C05472=1208.877,279.801,-65.738,-176.741,6.965,148.342
C05473=1208.880,279.552,-65.710,-176.743,6.963,148.342
C05474=1208.885,279.304,-65.681,-176.745,6.959,148.342
C05475=1208.889,279.056,-65.652,-176.748,6.958,148.342
C05476=1208.894,278.808,-65.624,-176.751,6.955,148.342
C05477=1208.898,278.559,-65.596,-176.753,6.952,148.342
C05478=1208.903,278.311,-65.567,-176.755,6.950,148.342
C05479=1208.907,278.063,-65.539,-176.758,6.947,148.342
C05480=1208.912,277.814,-65.511,-176.760,6.945,148.342
C05481=1208.915,277.566,-65.483,-176.763,6.942,148.343
C05482=1208.920,277.318,-65.455,-176.766,6.940,148.343
C05483=1208.924,277.069,-65.426,-176.768,6.938,148.343
C05484=1208.929,276.821,-65.398,-176.770,6.935,148.343
C05485=1208.933,276.572,-65.370,-176.773,6.933,148.343
C05486=1208.937,276.324,-65.342,-176.776,6.930,148.343
C05487=1208.941,276.076,-65.314,-176.778,6.928,148.343
C05488=1208.946,275.828,-65.285,-176.780,6.926,148.344
C05489=1208.950,275.579,-65.257,-176.783,6.923,148.344
C05490=1208.955,275.330,-65.230,-176.785,6.921,148.344
C05491=1208.959,275.082,-65.201,-176.788,6.918,148.344
C05492=1208.963,274.834,-65.174,-176.791,6.916,148.344
C05493=1208.968,274.585,-65.145,-176.793,6.914,148.344
C05494=1208.972,274.337,-65.117,-176.796,6.911,148.344
C05495=1208.976,274.088,-65.089,-176.798,6.909,148.344
C05496=1208.981,273.840,-65.061,-176.801,6.906,148.345
C05497=1208.985,273.592,-65.033,-176.803,6.904,148.345
C05498=1208.990,273.343,-65.005,-176.805,6.902,148.345
C05499=1208.995,273.095,-64.977,-176.809,6.899,148.345
C05500=1208.998,272.846,-64.949,-176.811,6.897,148.345
C05501=1209.003,272.599,-64.921,-176.813,6.895,148.345
C05502=1209.007,272.350,-64.893,-176.816,6.892,148.346
C05503=1209.012,272.101,-64.865,-176.818,6.890,148.346
C05504=1209.016,271.853,-64.837,-176.821,6.887,148.346
C05505=1209.020,271.605,-64.809,-176.824,6.885,148.346
C05506=1209.025,271.357,-64.781,-176.826,6.883,148.346
C05507=1209.029,271.107,-64.754,-176.829,6.880,148.346
C05508=1209.033,270.859,-64.726,-176.831,6.878,148.346
C05509=1209.038,270.612,-64.698,-176.834,6.876,148.347
C05510=1209.042,270.362,-64.671,-176.836,6.873,148.347
C05511=1209.047,270.114,-64.642,-176.838,6.871,148.347
C05512=1209.051,269.866,-64.614,-176.841,6.869,148.347
C05513=1209.055,269.617,-64.587,-176.844,6.866,148.347
C05514=1209.060,269.369,-64.559,-176.846,6.864,148.347
C05515=1209.064,269.120,-64.532,-176.849,6.861,148.347
C05516=1209.069,268.872,-64.504,-176.851,6.859,148.347
C05517=1209.073,268.624,-64.476,-176.854,6.857,148.348
C05518=1209.077,268.375,-64.448,-176.856,6.854,148.348
C05519=1209.082,268.127,-64.421,-176.859,6.852,148.348
C05520=1209.086,267.878,-64.393,-176.861,6.850,148.348
C05521=1209.090,267.630,-64.365,-176.864,6.847,148.348
C05522=1209.095,267.381,-64.338,-176.867,6.845,148.349
C05523=1209.100,267.133,-64.310,-176.869,6.843,148.349
C05524=1209.104,266.885,-64.282,-176.872,6.840,148.349
C05525=1209.108,266.636,-64.255,-176.874,6.838,148.349
C05526=1209.113,266.388,-64.228,-176.877,6.836,148.349
C05527=1209.117,266.139,-64.200,-176.879,6.833,148.349
C05528=1209.121,265.890,-64.172,-176.882,6.831,148.350
C05529=1209.126,265.643,-64.145,-176.884,6.829,148.350
C05530=1209.130,265.394,-64.118,-176.887,6.826,148.350
C05531=1209.134,265.146,-64.089,-176.889,6.824,148.350
C05532=1209.139,264.897,-64.062,-176.891,6.822,148.350
C05533=1209.144,264.649,-64.034,-176.895,6.819,148.350
C05534=1209.148,264.400,-64.007,-176.897,6.817,148.350
C05535=1209.152,264.151,-63.980,-176.899,6.815,148.351
C05536=1209.157,263.903,-63.952,-176.902,6.813,148.351
C05537=1209.161,263.655,-63.925,-176.905,6.810,148.351
C05538=1209.165,263.382,-63.895,-176.907,6.808,148.351
C05539=1209.171,263.109,-63.864,-176.910,6.806,148.351
C05540=1209.175,262.837,-63.835,-176.913,6.803,148.352
C05541=1209.180,262.564,-63.804,-176.915,6.801,148.352
C05542=1209.185,262.316,-63.777,-176.919,6.798,148.352
C05543=1209.189,262.067,-63.750,-176.921,6.796,148.352
C05544=1209.194,261.818,-63.723,-176.923,6.794,148.352
C05545=1209.198,261.570,-63.695,-176.926,6.791,148.352
C05546=1209.203,261.322,-63.668,-176.929,6.789,148.353
C05547=1209.207,261.072,-63.640,-176.931,6.787,148.353
C05548=1209.211,260.824,-63.614,-176.933,6.785,148.353
C05549=1209.215,260.576,-63.586,-176.936,6.782,148.353
C05550=1209.220,260.328,-63.559,-176.939,6.780,148.353
C05551=1209.224,260.079,-63.532,-176.941,6.778,148.354
C05552=1209.229,259.831,-63.505,-176.944,6.775,148.354
C05553=1209.233,259.582,-63.478,-176.946,6.773,148.354
C05554=1209.238,259.334,-63.450,-176.949,6.771,148.354
C05555=1209.242,259.085,-63.423,-176.951,6.769,148.354
C05556=1209.247,258.837,-63.396,-176.954,6.766,148.355
C05557=1209.251,258.589,-63.369,-176.956,6.764,148.355
C05558=1209.255,258.340,-63.342,-176.959,6.762,148.355
C05559=1209.259,258.091,-63.315,-176.962,6.759,148.355
C05560=1209.264,257.842,-63.288,-176.964,6.757,148.355
C05561=1209.269,257.594,-63.261,-176.966,6.755,148.355
C05562=1209.273,257.346,-63.234,-176.969,6.753,148.356
C05563=1209.277,257.097,-63.207,-176.972,6.750,148.356
C05564=1209.282,256.849,-63.180,-176.974,6.748,148.356
C05565=1209.287,256.600,-63.153,-176.976,6.746,148.356
C05566=1209.291,256.351,-63.126,-176.979,6.744,148.356
C05567=1209.295,256.103,-63.098,-176.982,6.741,148.356
C05568=1209.299,255.854,-63.072,-176.984,6.740,148.357
C05569=1209.304,255.606,-63.045,-176.987,6.738,148.357
C05570=1209.309,255.357,-63.018,-176.989,6.735,148.357
C05571=1209.313,255.109,-62.991,-176.992,6.733,148.357
C05572=1209.317,254.861,-62.964,-176.994,6.731,148.358
C05573=1209.322,254.612,-62.937,-176.997,6.729,148.358
C05574=1209.327,254.364,-62.910,-177.000,6.726,148.358
C05575=1209.331,254.115,-62.883,-177.002,6.724,148.358
C05576=1209.335,253.867,-62.857,-177.004,6.722,148.358
C05577=1209.340,253.619,-62.830,-177.007,6.720,148.359
C05578=1209.344,253.369,-62.802,-177.010,6.718,148.359
C05579=1209.348,253.121,-62.776,-177.012,6.715,148.359
C05580=1209.352,252.873,-62.749,-177.015,6.713,148.359
C05581=1209.357,252.624,-62.722,-177.017,6.711,148.359
C05582=1209.361,252.375,-62.696,-177.020,6.709,148.360
C05583=1209.366,252.127,-62.669,-177.022,6.706,148.360
C05584=1209.371,251.878,-62.642,-177.025,6.704,148.360
C05585=1209.375,251.630,-62.615,-177.028,6.702,148.360
C05586=1209.379,251.381,-62.589,-177.030,6.700,148.360
C05587=1209.384,251.133,-62.562,-177.033,6.697,148.361
C05588=1209.388,250.884,-62.535,-177.035,6.695,148.361
C05589=1209.393,250.636,-62.508,-177.038,6.693,148.361
C05590=1209.397,250.387,-62.483,-177.040,6.691,148.361
C05591=1209.402,250.139,-62.456,-177.043,6.689,148.361
C05592=1209.406,249.890,-62.429,-177.046,6.687,148.362
C05593=1209.410,249.642,-62.402,-177.048,6.684,148.362
C05594=1209.415,249.393,-62.376,-177.051,6.683,148.362
C05595=1209.419,249.145,-62.349,-177.053,6.680,148.362
C05596=1209.424,248.896,-62.322,-177.056,6.678,148.363
C05597=1209.428,248.647,-62.296,-177.058,6.676,148.363
C05598=1209.433,248.399,-62.269,-177.061,6.674,148.363
C05599=1209.436,248.151,-62.243,-177.063,6.672,148.363
C05600=1209.441,247.902,-62.217,-177.065,6.670,148.363
C05601=1209.446,247.653,-62.189,-177.069,6.667,148.364
C05602=1209.450,247.404,-62.164,-177.071,6.665,148.364
C05603=1209.455,247.156,-62.137,-177.073,6.663,148.364
C05604=1209.460,246.908,-62.111,-177.076,6.661,148.364
C05605=1209.464,246.659,-62.084,-177.078,6.659,148.364
C05606=1209.468,246.411,-62.058,-177.081,6.656,148.365
C05607=1209.473,246.162,-62.031,-177.084,6.654,148.365
C05608=1209.477,245.914,-62.005,-177.086,6.652,148.365
C05609=1209.482,245.665,-61.979,-177.089,6.650,148.365
C05610=1209.486,245.416,-61.952,-177.091,6.648,148.366
C05611=1209.490,245.168,-61.926,-177.094,6.645,148.366
C05612=1209.495,244.919,-61.899,-177.097,6.644,148.366
C05613=1209.499,244.670,-61.874,-177.099,6.642,148.366
C05614=1209.504,244.422,-61.847,-177.101,6.640,148.367
C05615=1209.508,244.173,-61.821,-177.104,6.638,148.367
C05616=1209.513,243.926,-61.795,-177.107,6.635,148.367
C05617=1209.518,243.676,-61.768,-177.109,6.633,148.367
C05618=1209.522,243.428,-61.743,-177.112,6.631,148.368
C05619=1209.527,243.179,-61.715,-177.114,6.629,148.368
C05620=1209.531,242.930,-61.690,-177.117,6.627,148.368
C05621=1209.535,242.682,-61.663,-177.119,6.625,148.368
C05622=1209.540,242.433,-61.637,-177.122,6.622,148.368
C05623=1209.544,242.185,-61.612,-177.125,6.620,148.369
C05624=1209.548,241.937,-61.585,-177.127,6.618,148.369
C05625=1209.553,241.688,-61.559,-177.129,6.616,148.369
C05626=1209.558,241.439,-61.533,-177.132,6.614,148.369
C05627=1209.561,241.191,-61.507,-177.135,6.613,148.370
C05628=1209.566,240.941,-61.480,-177.137,6.609,148.370
C05629=1209.571,240.693,-61.455,-177.140,6.608,148.370
C05630=1209.575,240.445,-61.429,-177.143,6.606,148.370
C05631=1209.580,240.196,-61.402,-177.145,6.604,148.370
C05632=1209.584,239.947,-61.376,-177.147,6.602,148.371
C05633=1209.589,239.698,-61.350,-177.150,6.600,148.371
C05634=1209.593,239.450,-61.325,-177.153,6.597,148.371
C05635=1209.598,239.202,-61.298,-177.155,6.595,148.371
C05636=1209.602,238.953,-61.272,-177.158,6.593,148.372
C05637=1209.607,238.704,-61.247,-177.160,6.591,148.372
C05638=1209.611,238.455,-61.221,-177.163,6.589,148.372
C05639=1209.616,238.207,-61.195,-177.165,6.587,148.372
C05640=1209.620,237.959,-61.168,-177.168,6.585,148.373
C05641=1209.624,237.710,-61.143,-177.171,6.582,148.373
C05642=1209.629,237.438,-61.115,-177.173,6.581,148.373
C05643=1209.634,237.168,-61.086,-177.176,6.579,148.374
C05644=1209.640,236.895,-61.058,-177.179,6.576,148.374
C05645=1209.645,236.624,-61.030,-177.182,6.574,148.374
C05646=1209.649,236.375,-61.004,-177.184,6.572,148.374
C05647=1209.653,236.127,-60.978,-177.187,6.569,148.374
C05648=1209.657,235.878,-60.952,-177.190,6.568,148.375
C05649=1209.662,235.630,-60.926,-177.192,6.565,148.375
C05650=1209.666,235.381,-60.901,-177.195,6.563,148.375
C05651=1209.671,235.132,-60.874,-177.197,6.562,148.376
C05652=1209.675,234.884,-60.849,-177.200,6.560,148.376
C05653=1209.680,234.635,-60.823,-177.202,6.558,148.376
C05654=1209.685,234.387,-60.798,-177.205,6.556,148.376
C05655=1209.689,234.138,-60.772,-177.208,6.553,148.377
C05656=1209.694,233.890,-60.746,-177.210,6.551,148.377
C05657=1209.698,233.641,-60.721,-177.213,6.549,148.377
C05658=1209.702,233.392,-60.695,-177.215,6.547,148.377
C05659=1209.707,233.144,-60.669,-177.218,6.545,148.378
C05660=1209.712,232.895,-60.643,-177.220,6.543,148.378
C05661=1209.716,232.645,-60.618,-177.223,6.541,148.378
C05662=1209.721,232.397,-60.592,-177.225,6.539,148.378
C05663=1209.725,232.149,-60.567,-177.228,6.538,148.379
C05664=1209.730,231.900,-60.541,-177.231,6.535,148.379
C05665=1209.734,231.652,-60.516,-177.233,6.533,148.379
C05666=1209.739,231.403,-60.490,-177.236,6.531,148.379
C05667=1209.743,231.154,-60.464,-177.239,6.529,148.380
C05668=1209.748,230.906,-60.439,-177.241,6.527,148.380
C05669=1209.752,230.657,-60.414,-177.243,6.525,148.380
C05670=1209.756,230.408,-60.388,-177.246,6.523,148.380
C05671=1209.761,230.160,-60.363,-177.249,6.521,148.381
C05672=1209.766,229.911,-60.337,-177.251,6.519,148.381
C05673=1209.770,229.662,-60.311,-177.253,6.517,148.381
C05674=1209.775,229.413,-60.287,-177.257,6.515,148.382
C05675=1209.779,229.164,-60.261,-177.259,6.513,148.382
C05676=1209.784,228.916,-60.235,-177.262,6.511,148.382
C05677=1209.788,228.668,-60.210,-177.264,6.509,148.382
C05678=1209.793,228.418,-60.185,-177.267,6.507,148.383
C05679=1209.798,228.170,-60.159,-177.269,6.505,148.383
C05680=1209.801,227.922,-60.134,-177.272,6.503,148.383
C05681=1209.806,227.673,-60.109,-177.274,6.501,148.383
C05682=1209.810,227.424,-60.084,-177.277,6.499,148.384
C05683=1209.815,227.175,-60.058,-177.279,6.497,148.384
C05684=1209.819,226.927,-60.033,-177.282,6.496,148.384
C05685=1209.824,226.678,-60.008,-177.285,6.493,148.385
C05686=1209.829,226.430,-59.982,-177.287,6.491,148.385
C05687=1209.833,226.181,-59.956,-177.290,6.489,148.385
C05688=1209.838,225.932,-59.932,-177.293,6.487,148.385
C05689=1209.842,225.684,-59.907,-177.295,6.485,148.386
C05690=1209.847,225.435,-59.882,-177.298,6.483,148.386
C05691=1209.851,225.186,-59.856,-177.300,6.481,148.386
C05692=1209.856,224.938,-59.831,-177.303,6.479,148.386
C05693=1209.860,224.689,-59.806,-177.305,6.477,148.387
C05694=1209.865,224.440,-59.780,-177.308,6.476,148.387
C05695=1209.869,224.191,-59.756,-177.310,6.474,148.387
C05696=1209.873,223.942,-59.730,-177.313,6.472,148.388
C05697=1209.878,223.694,-59.705,-177.315,6.470,148.388
C05698=1209.883,223.445,-59.680,-177.318,6.468,148.388
C05699=1209.888,223.196,-59.655,-177.321,6.465,148.388
C05700=1209.891,222.948,-59.630,-177.324,6.463,148.389
C05701=1209.896,222.699,-59.605,-177.326,6.461,148.389
C05702=1209.900,222.450,-59.580,-177.329,6.459,148.389
C05703=1209.906,222.201,-59.555,-177.331,6.458,148.390
C05704=1209.909,221.953,-59.530,-177.334,6.456,148.390
C05705=1209.914,221.704,-59.505,-177.336,6.454,148.390
C05706=1209.919,221.456,-59.480,-177.339,6.452,148.391
C05707=1209.924,221.207,-59.455,-177.341,6.450,148.391
C05708=1209.928,220.958,-59.431,-177.344,6.448,148.391
C05709=1209.932,220.710,-59.405,-177.347,6.446,148.391
C05710=1209.937,220.461,-59.380,-177.349,6.444,148.392
C05711=1209.941,220.212,-59.356,-177.352,6.442,148.392
C05712=1209.946,219.964,-59.330,-177.354,6.441,148.392
C05713=1209.950,219.714,-59.305,-177.357,6.439,148.393
C05714=1209.955,219.466,-59.281,-177.359,6.437,148.393
C05715=1209.959,219.217,-59.255,-177.362,6.435,148.393
C05716=1209.964,218.968,-59.231,-177.364,6.433,148.393
C05717=1209.969,218.720,-59.207,-177.368,6.430,148.394
C05718=1209.973,218.471,-59.181,-177.370,6.428,148.394
C05719=1209.978,218.222,-59.156,-177.373,6.427,148.394
C05720=1209.982,217.973,-59.132,-177.376,6.425,148.395
C05721=1209.987,217.724,-59.107,-177.378,6.423,148.395
C05722=1209.991,217.477,-59.082,-177.380,6.421,148.395
C05723=1209.996,217.227,-59.057,-177.383,6.419,148.395
C05724=1210.001,216.979,-59.033,-177.386,6.417,148.396
C05725=1210.004,216.729,-59.008,-177.388,6.415,148.396
C05726=1210.010,216.481,-58.984,-177.391,6.413,148.396
C05727=1210.014,216.233,-58.959,-177.394,6.412,148.397
C05728=1210.018,215.983,-58.934,-177.396,6.409,148.397
C05729=1210.023,215.735,-58.909,-177.398,6.408,148.397
C05730=1210.028,215.486,-58.885,-177.401,6.406,148.398
C05731=1210.032,215.237,-58.860,-177.404,6.404,148.398
C05732=1210.037,214.988,-58.836,-177.406,6.402,148.398
C05733=1210.041,214.740,-58.810,-177.409,6.400,148.399
C05734=1210.045,214.491,-58.786,-177.412,6.398,148.399
C05735=1210.050,214.243,-58.761,-177.414,6.396,148.399
C05736=1210.055,213.994,-58.737,-177.417,6.395,148.400
C05737=1210.059,213.745,-58.712,-177.420,6.393,148.400
C05738=1210.064,213.496,-58.688,-177.422,6.391,148.400
C05739=1210.069,213.248,-58.663,-177.424,6.389,148.400
C05740=1210.073,212.998,-58.639,-177.427,6.387,148.401
C05741=1210.078,212.750,-58.614,-177.430,6.385,148.401
C05742=1210.082,212.501,-58.590,-177.432,6.383,148.401
C05743=1210.087,212.252,-58.565,-177.435,6.381,148.402
C05744=1210.091,212.003,-58.541,-177.438,6.380,148.402
C05745=1210.096,211.755,-58.517,-177.440,6.378,148.402
C05746=1210.101,211.485,-58.490,-177.443,6.375,148.403
C05747=1210.105,211.214,-58.463,-177.446,6.373,148.403
C05748=1210.111,210.943,-58.437,-177.449,6.371,148.403
C05749=1210.116,210.673,-58.411,-177.451,6.370,148.404
C05750=1210.120,210.425,-58.387,-177.454,6.368,148.404
C05751=1210.125,210.175,-58.362,-177.457,6.366,148.404
C05752=1210.129,209.927,-58.337,-177.459,6.364,148.405
C05753=1210.134,209.678,-58.313,-177.462,6.362,148.405
C05754=1210.139,209.430,-58.289,-177.464,6.360,148.405
C05755=1210.142,209.181,-58.264,-177.467,6.359,148.406
C05756=1210.147,208.932,-58.241,-177.470,6.357,148.406
C05757=1210.152,208.683,-58.216,-177.472,6.355,148.406
C05758=1210.157,208.434,-58.192,-177.475,6.353,148.407
C05759=1210.160,208.185,-58.168,-177.477,6.351,148.407
C05760=1210.166,207.937,-58.143,-177.480,6.349,148.407
C05761=1210.170,207.688,-58.119,-177.483,6.347,148.408
C05762=1210.175,207.439,-58.096,-177.485,6.345,148.408
C05763=1210.180,207.190,-58.071,-177.488,6.344,148.408
C05764=1210.184,206.941,-58.047,-177.490,6.342,148.409
C05765=1210.188,206.693,-58.022,-177.493,6.340,148.409
C05766=1210.193,206.444,-57.998,-177.496,6.338,148.409
C05767=1210.198,206.195,-57.974,-177.498,6.336,148.410
C05768=1210.202,205.947,-57.950,-177.501,6.334,148.410
C05769=1210.207,205.698,-57.926,-177.504,6.333,148.410
C05770=1210.211,205.448,-57.902,-177.506,6.331,148.411
C05771=1210.216,205.200,-57.878,-177.509,6.329,148.411
C05772=1210.220,204.951,-57.854,-177.512,6.327,148.411
C05773=1210.225,204.702,-57.830,-177.514,6.325,148.412
C05774=1210.230,204.454,-57.806,-177.517,6.323,148.412
C05775=1210.234,204.205,-57.781,-177.519,6.321,148.412
C05776=1210.239,203.956,-57.758,-177.522,6.319,148.412
C05777=1210.243,203.707,-57.734,-177.524,6.318,148.413
C05778=1210.247,203.459,-57.710,-177.527,6.316,148.413
C05779=1210.253,203.209,-57.686,-177.530,6.314,148.413
C05780=1210.257,202.961,-57.662,-177.532,6.313,148.414
C05781=1210.262,202.712,-57.638,-177.534,6.311,148.414
C05782=1210.266,202.464,-57.614,-177.537,6.309,148.414
C05783=1210.270,202.214,-57.591,-177.540,6.307,148.415
C05784=1210.275,201.965,-57.567,-177.542,6.306,148.415
C05785=1210.280,201.717,-57.542,-177.545,6.304,148.415
C05786=1210.285,201.468,-57.519,-177.548,6.302,148.416
C05787=1210.289,201.219,-57.494,-177.550,6.300,148.416
C05788=1210.294,200.970,-57.471,-177.553,6.298,148.417
C05789=1210.298,200.722,-57.447,-177.556,6.296,148.417
C05790=1210.303,200.473,-57.424,-177.558,6.295,148.417
C05791=1210.307,200.224,-57.400,-177.561,6.293,148.418
C05792=1210.312,199.975,-57.376,-177.563,6.291,148.418
C05793=1210.316,199.726,-57.352,-177.566,6.289,148.418
C05794=1210.321,199.477,-57.328,-177.569,6.287,148.419
C05795=1210.326,199.228,-57.304,-177.571,6.286,148.419
C05796=1210.330,198.979,-57.280,-177.573,6.284,148.419
C05797=1210.335,198.730,-57.257,-177.576,6.283,148.420
C05798=1210.339,198.482,-57.233,-177.579,6.281,148.420
C05799=1210.344,198.233,-57.210,-177.581,6.279,148.420
C05800=1210.349,197.984,-57.186,-177.584,6.277,148.421
C05801=1210.353,197.735,-57.162,-177.587,6.275,148.421
C05802=1210.358,197.486,-57.139,-177.589,6.273,148.421
C05803=1210.363,197.237,-57.115,-177.592,6.272,148.422
C05804=1210.367,196.989,-57.091,-177.595,6.270,148.422
C05805=1210.372,196.740,-57.068,-177.597,6.268,148.422
C05806=1210.376,196.491,-57.045,-177.600,6.266,148.423
C05807=1210.381,196.242,-57.021,-177.602,6.265,148.423
C05808=1210.385,195.993,-56.997,-177.605,6.263,148.423
C05809=1210.390,195.744,-56.974,-177.607,6.262,148.424
C05810=1210.394,195.496,-56.950,-177.610,6.260,148.424
C05811=1210.399,195.247,-56.926,-177.613,6.258,148.424
C05812=1210.404,194.998,-56.903,-177.615,6.256,148.425
C05813=1210.409,194.749,-56.880,-177.618,6.254,148.425
C05814=1210.413,194.500,-56.856,-177.621,6.252,148.426
C05815=1210.418,194.251,-56.832,-177.623,6.251,148.426
C05816=1210.422,194.002,-56.809,-177.625,6.250,148.426
C05817=1210.426,193.754,-56.786,-177.628,6.248,148.427
C05818=1210.431,193.505,-56.763,-177.631,6.246,148.427
C05819=1210.435,193.256,-56.739,-177.633,6.244,148.427
C05820=1210.440,193.007,-56.715,-177.636,6.242,148.428
C05821=1210.445,192.758,-56.692,-177.639,6.240,148.428
C05822=1210.450,192.509,-56.669,-177.641,6.239,148.428
C05823=1210.455,192.261,-56.646,-177.644,6.237,148.429
C05824=1210.460,192.012,-56.622,-177.646,6.236,148.429
C05825=1210.464,191.763,-56.599,-177.649,6.234,148.430
C05826=1210.468,191.514,-56.576,-177.652,6.232,148.430
C05827=1210.473,191.266,-56.552,-177.654,6.231,148.430
C05828=1210.477,191.017,-56.529,-177.657,6.229,148.431
C05829=1210.482,190.768,-56.505,-177.660,6.227,148.431
C05830=1210.487,190.519,-56.482,-177.662,6.225,148.431
C05831=1210.491,190.270,-56.459,-177.665,6.223,148.432
C05832=1210.495,190.021,-56.436,-177.667,6.222,148.432
C05833=1210.500,189.772,-56.413,-177.670,6.221,148.432
C05834=1210.505,189.523,-56.390,-177.672,6.219,148.433
C05835=1210.510,189.274,-56.366,-177.675,6.217,148.433
C05836=1210.514,189.026,-56.343,-177.678,6.215,148.434
C05837=1210.519,188.777,-56.320,-177.680,6.213,148.434
C05838=1210.523,188.528,-56.297,-177.683,6.211,148.434
C05839=1210.528,188.279,-56.273,-177.685,6.210,148.435
C05840=1210.533,188.030,-56.250,-177.688,6.209,148.435
C05841=1210.537,187.781,-56.227,-177.690,6.207,148.435
C05842=1210.542,187.532,-56.204,-177.694,6.205,148.436
C05843=1210.547,187.283,-56.182,-177.696,6.203,148.436
C05844=1210.551,187.034,-56.159,-177.699,6.202,148.437
C05845=1210.556,186.785,-56.135,-177.701,6.201,148.437
C05846=1210.560,186.536,-56.112,-177.704,6.199,148.437
C05847=1210.565,186.287,-56.089,-177.706,6.197,148.438
C05848=1210.570,186.039,-56.066,-177.709,6.195,148.438
C05849=1210.574,185.790,-56.043,-177.712,6.193,148.438
C05850=1210.580,185.520,-56.018,-177.714,6.192,148.439
C05851=1210.584,185.251,-55.994,-177.717,6.190,148.439
C05852=1210.590,184.981,-55.968,-177.720,6.188,148.440
C05853=1210.594,184.712,-55.944,-177.723,6.186,148.440
C05854=1210.599,184.462,-55.921,-177.725,6.185,148.440
C05855=1210.604,184.213,-55.897,-177.728,6.183,148.441
C05856=1210.608,183.964,-55.875,-177.731,6.181,148.441
C05857=1210.613,183.716,-55.852,-177.733,6.180,148.441
C05858=1210.618,183.467,-55.829,-177.736,6.178,148.442
C05859=1210.622,183.218,-55.806,-177.739,6.177,148.442
C05860=1210.627,182.968,-55.784,-177.741,6.175,148.443
C05861=1210.631,182.720,-55.761,-177.744,6.173,148.443
C05862=1210.636,182.471,-55.738,-177.746,6.172,148.443
C05863=1210.641,182.222,-55.714,-177.749,6.170,148.444
C05864=1210.645,181.973,-55.692,-177.751,6.168,148.444
C05865=1210.650,181.724,-55.669,-177.754,6.167,148.445
C05866=1210.654,181.476,-55.647,-177.757,6.165,148.445
C05867=1210.659,181.226,-55.624,-177.759,6.164,148.445
C05868=1210.663,180.978,-55.601,-177.762,6.162,148.446
C05869=1210.668,180.728,-55.578,-177.764,6.160,148.446
C05870=1210.673,180.480,-55.556,-177.767,6.159,148.447
C05871=1210.678,180.231,-55.533,-177.770,6.157,148.447
C05872=1210.682,179.981,-55.511,-177.772,6.156,148.447
C05873=1210.687,179.733,-55.488,-177.775,6.154,148.448
C05874=1210.691,179.484,-55.465,-177.777,6.152,148.448
C05875=1210.696,179.235,-55.442,-177.780,6.150,148.448
C05876=1210.701,178.987,-55.420,-177.783,6.149,148.449
C05877=1210.706,178.737,-55.397,-177.785,6.148,148.449
C05878=1210.710,178.488,-55.375,-177.788,6.146,148.450
C05879=1210.715,178.239,-55.352,-177.790,6.144,148.450
C05880=1210.719,177.991,-55.329,-177.793,6.142,148.450
C05881=1210.724,177.741,-55.307,-177.795,6.141,148.451
C05882=1210.728,177.492,-55.284,-177.798,6.140,148.451
C05883=1210.734,177.243,-55.262,-177.801,6.138,148.451
C05884=1210.738,176.995,-55.239,-177.804,6.136,148.452
C05885=1210.742,176.745,-55.217,-177.806,6.135,148.452
C05886=1210.747,176.497,-55.194,-177.808,6.134,148.453
C05887=1210.752,176.248,-55.172,-177.811,6.132,148.453
C05888=1210.756,175.999,-55.149,-177.814,6.130,148.454
C05889=1210.761,175.750,-55.127,-177.816,6.128,148.454
C05890=1210.765,175.501,-55.104,-177.818,6.127,148.454
C05891=1210.771,175.252,-55.082,-177.822,6.126,148.455
C05892=1210.775,175.003,-55.060,-177.824,6.124,148.455
C05893=1210.780,174.754,-55.036,-177.827,6.122,148.456
C05894=1210.785,174.505,-55.015,-177.829,6.121,148.456
C05895=1210.789,174.257,-54.992,-177.832,6.119,148.456
C05896=1210.794,174.007,-54.969,-177.834,6.117,148.457
C05897=1210.798,173.758,-54.948,-177.838,6.116,148.457
C05898=1210.802,173.510,-54.925,-177.840,6.115,148.458
C05899=1210.808,173.261,-54.903,-177.842,6.113,148.458
C05900=1210.812,173.011,-54.881,-177.845,6.111,148.458
C05901=1210.817,172.763,-54.858,-177.848,6.109,148.459
C05902=1210.822,172.514,-54.836,-177.850,6.109,148.459
C05903=1210.826,172.264,-54.814,-177.853,6.107,148.460
C05904=1210.831,172.016,-54.792,-177.855,6.105,148.460
C05905=1210.836,171.767,-54.768,-177.858,6.103,148.460
C05906=1210.841,171.518,-54.747,-177.860,6.102,148.461
C05907=1210.845,171.269,-54.725,-177.863,6.101,148.461
C05908=1210.850,171.020,-54.703,-177.866,6.099,148.462
C05909=1210.854,170.771,-54.680,-177.869,6.097,148.462
C05910=1210.859,170.522,-54.658,-177.871,6.096,148.463
C05911=1210.863,170.273,-54.636,-177.873,6.095,148.463
C05912=1210.868,170.024,-54.614,-177.876,6.093,148.463
C05913=1210.873,169.775,-54.592,-177.879,6.091,148.464
C05914=1210.878,169.525,-54.570,-177.881,6.090,148.464
C05915=1210.882,169.277,-54.547,-177.884,6.088,148.465
C05916=1210.886,169.028,-54.525,-177.887,6.087,148.465
C05917=1210.891,168.779,-54.503,-177.889,6.086,148.465
C05918=1210.896,168.530,-54.481,-177.891,6.084,148.466
C05919=1210.901,168.281,-54.459,-177.894,6.082,148.466
C05920=1210.905,168.032,-54.437,-177.897,6.081,148.467
C05921=1210.910,167.783,-54.415,-177.899,6.080,148.467
C05922=1210.915,167.534,-54.393,-177.902,6.078,148.467
C05923=1210.920,167.285,-54.370,-177.905,6.076,148.468
C05924=1210.924,167.036,-54.348,-177.907,6.075,148.468
C05925=1210.929,166.787,-54.327,-177.910,6.074,148.469
C05926=1210.933,166.538,-54.305,-177.913,6.072,148.469
C05927=1210.938,166.289,-54.283,-177.915,6.070,148.469
C05928=1210.942,166.040,-54.261,-177.917,6.069,148.470
C05929=1210.947,165.791,-54.239,-177.920,6.067,148.470
C05930=1210.952,165.542,-54.217,-177.923,6.066,148.471
C05931=1210.956,165.293,-54.195,-177.925,6.065,148.471
C05932=1210.962,165.044,-54.173,-177.928,6.063,148.472
C05933=1210.966,164.795,-54.151,-177.931,6.061,148.472
C05934=1210.971,164.547,-54.129,-177.933,6.060,148.472
C05935=1210.975,164.297,-54.107,-177.936,6.059,148.473
C05936=1210.980,164.049,-54.086,-177.939,6.057,148.473
C05937=1210.985,163.799,-54.064,-177.941,6.056,148.474
C05938=1210.990,163.550,-54.043,-177.943,6.054,148.474
C05939=1210.994,163.301,-54.021,-177.946,6.053,148.475
C05940=1210.999,163.052,-53.999,-177.949,6.051,148.475
C05941=1211.004,162.803,-53.977,-177.951,6.050,148.475
C05942=1211.008,162.554,-53.955,-177.954,6.048,148.476
C05943=1211.013,162.305,-53.934,-177.957,6.046,148.476
C05944=1211.017,162.056,-53.912,-177.959,6.045,148.477
C05945=1211.022,161.807,-53.890,-177.962,6.044,148.477
C05946=1211.027,161.558,-53.869,-177.965,6.042,148.477
C05947=1211.032,161.309,-53.847,-177.967,6.041,148.478
C05948=1211.036,161.060,-53.825,-177.970,6.039,148.478
C05949=1211.041,160.811,-53.803,-177.972,6.038,148.479
C05950=1211.046,160.562,-53.781,-177.975,6.037,148.479
C05951=1211.050,160.313,-53.760,-177.977,6.035,148.480
C05952=1211.055,160.064,-53.738,-177.980,6.033,148.480
C05953=1211.060,159.815,-53.717,-177.982,6.032,148.481
C05954=1211.065,159.546,-53.693,-177.985,6.031,148.481
C05955=1211.070,159.277,-53.670,-177.988,6.029,148.482
C05956=1211.075,159.008,-53.647,-177.991,6.027,148.482
C05957=1211.080,158.739,-53.624,-177.994,6.026,148.483
C05958=1211.085,158.490,-53.602,-177.996,6.025,148.483
C05959=1211.089,158.241,-53.580,-177.999,6.023,148.483
C05960=1211.094,157.991,-53.559,-178.002,6.021,148.484
C05961=1211.099,157.743,-53.537,-178.004,6.021,148.484
C05962=1211.103,157.493,-53.515,-178.007,6.019,148.485
C05963=1211.109,157.244,-53.494,-178.009,6.017,148.485
C05964=1211.113,156.996,-53.473,-178.012,6.016,148.485
C05965=1211.117,156.747,-53.451,-178.015,6.015,148.486
C05966=1211.122,156.497,-53.430,-178.017,6.013,148.486
C05967=1211.127,156.249,-53.409,-178.020,6.012,148.487
C05968=1211.132,156.000,-53.387,-178.023,6.010,148.487
C05969=1211.137,155.750,-53.366,-178.025,6.009,148.488
C05970=1211.141,155.501,-53.344,-178.027,6.008,148.488
C05971=1211.146,155.252,-53.323,-178.030,6.006,148.488
C05972=1211.150,155.003,-53.301,-178.033,6.005,148.489
C05973=1211.155,154.754,-53.280,-178.035,6.003,148.489
C05974=1211.160,154.505,-53.259,-178.038,6.002,148.490
C05975=1211.165,154.257,-53.237,-178.040,6.001,148.490
C05976=1211.169,154.007,-53.216,-178.043,5.999,148.491
C05977=1211.174,153.758,-53.195,-178.046,5.997,148.491
C05978=1211.179,153.509,-53.174,-178.048,5.996,148.492
C05979=1211.184,153.260,-53.152,-178.051,5.995,148.492
C05980=1211.188,153.011,-53.131,-178.053,5.994,148.493
C05981=1211.192,152.762,-53.110,-178.056,5.992,148.493
C05982=1211.198,152.513,-53.089,-178.059,5.990,148.493
C05983=1211.202,152.264,-53.067,-178.061,5.990,148.494
C05984=1211.207,152.015,-53.047,-178.064,5.988,148.494
C05985=1211.211,151.765,-53.025,-178.066,5.987,148.495
C05986=1211.216,151.517,-53.004,-178.069,5.985,148.495
C05987=1211.222,151.267,-52.983,-178.072,5.984,148.496
C05988=1211.226,151.019,-52.962,-178.074,5.983,148.496
C05989=1211.231,150.770,-52.941,-178.077,5.981,148.497
C05990=1211.235,150.520,-52.919,-178.079,5.980,148.497
C05991=1211.240,150.271,-52.898,-178.082,5.978,148.497
C05992=1211.245,150.022,-52.877,-178.085,5.977,148.498
C05993=1211.250,149.774,-52.855,-178.087,5.976,148.498
C05994=1211.254,149.525,-52.835,-178.090,5.974,148.499
C05995=1211.259,149.275,-52.814,-178.092,5.973,148.499
C05996=1211.263,149.026,-52.792,-178.095,5.972,148.500
C05997=1211.268,148.777,-52.772,-178.098,5.970,148.500
C05998=1211.273,148.528,-52.751,-178.100,5.969,148.501
C05999=1211.278,148.279,-52.729,-178.103,5.968,148.501
C06000=1211.282,148.030,-52.709,-178.105,5.967,148.502
C06001=1211.287,147.780,-52.687,-178.108,5.965,148.502
C06002=1211.292,147.531,-52.666,-178.111,5.963,148.503
C06003=1211.296,147.283,-52.645,-178.113,5.962,148.503
C06004=1211.301,147.033,-52.624,-178.116,5.961,148.503
C06005=1211.306,146.784,-52.604,-178.118,5.960,148.504
C06006=1211.311,146.535,-52.583,-178.121,5.958,148.504
C06007=1211.316,146.287,-52.561,-178.123,5.957,148.505
C06008=1211.320,146.038,-52.541,-178.126,5.956,148.505
C06009=1211.325,145.788,-52.520,-178.129,5.954,148.506
C06010=1211.329,145.539,-52.499,-178.131,5.953,148.506
C06011=1211.335,145.289,-52.478,-178.134,5.951,148.507
C06012=1211.339,145.041,-52.457,-178.136,5.951,148.507
C06013=1211.344,144.792,-52.436,-178.139,5.949,148.508
C06014=1211.348,144.543,-52.416,-178.142,5.948,148.508
C06015=1211.353,144.294,-52.395,-178.144,5.946,148.509
C06016=1211.358,144.045,-52.375,-178.147,5.945,148.509
C06017=1211.363,143.795,-52.354,-178.150,5.944,148.510
C06018=1211.368,143.547,-52.333,-178.152,5.942,148.510
C06019=1211.372,143.297,-52.312,-178.154,5.941,148.510
C06020=1211.376,143.048,-52.291,-178.158,5.940,148.511
C06021=1211.381,142.799,-52.270,-178.160,5.939,148.511
C06022=1211.386,142.550,-52.249,-178.162,5.937,148.512
C06023=1211.391,142.301,-52.228,-178.165,5.936,148.512
C06024=1211.395,142.052,-52.208,-178.168,5.934,148.513
C06025=1211.401,141.803,-52.187,-178.170,5.933,148.513
C06026=1211.405,141.554,-52.167,-178.173,5.932,148.514
C06027=1211.410,141.304,-52.146,-178.176,5.930,148.514
C06028=1211.415,141.055,-52.125,-178.178,5.929,148.515
C06029=1211.419,140.806,-52.105,-178.181,5.928,148.515
C06030=1211.424,140.557,-52.084,-178.183,5.927,148.516
C06031=1211.429,140.308,-52.064,-178.186,5.925,148.516
C06032=1211.434,140.059,-52.043,-178.188,5.924,148.517
C06033=1211.438,139.810,-52.022,-178.191,5.923,148.517
C06034=1211.443,139.561,-52.002,-178.194,5.922,148.518
C06035=1211.448,139.312,-51.981,-178.196,5.920,148.518
C06036=1211.452,139.063,-51.961,-178.198,5.919,148.518
C06037=1211.458,138.814,-51.940,-178.202,5.918,148.519
C06038=1211.462,138.565,-51.919,-178.204,5.916,148.519
C06039=1211.467,138.315,-51.900,-178.207,5.915,148.520
C06040=1211.472,138.066,-51.879,-178.209,5.914,148.520
C06041=1211.476,137.817,-51.858,-178.212,5.913,148.521
C06042=1211.481,137.568,-51.838,-178.215,5.911,148.521
C06043=1211.486,137.319,-51.817,-178.217,5.910,148.522
C06044=1211.490,137.070,-51.797,-178.220,5.908,148.522
C06045=1211.495,136.821,-51.776,-178.222,5.908,148.523
C06046=1211.500,136.571,-51.756,-178.225,5.906,148.523
C06047=1211.505,136.322,-51.736,-178.227,5.905,148.524
C06048=1211.509,136.073,-51.715,-178.230,5.904,148.524
C06049=1211.514,135.824,-51.694,-178.232,5.903,148.525
C06050=1211.519,135.575,-51.674,-178.235,5.901,148.525
C06051=1211.524,135.325,-51.654,-178.238,5.900,148.526
C06052=1211.528,135.076,-51.634,-178.241,5.899,148.526
C06053=1211.534,134.828,-51.613,-178.243,5.898,148.527
C06054=1211.538,134.579,-51.593,-178.245,5.896,148.527
C06055=1211.543,134.330,-51.573,-178.248,5.895,148.528
C06056=1211.548,134.080,-51.552,-178.251,5.894,148.528
C06057=1211.553,133.831,-51.532,-178.253,5.893,148.529
C06058=1211.557,133.562,-51.511,-178.256,5.891,148.529
C06059=1211.563,133.294,-51.488,-178.259,5.890,148.530
C06060=1211.568,133.024,-51.466,-178.261,5.889,148.530
C06061=1211.572,132.756,-51.445,-178.264,5.887,148.531
C06062=1211.577,132.507,-51.424,-178.267,5.886,148.531
C06063=1211.583,132.258,-51.404,-178.270,5.885,148.532
C06064=1211.587,132.009,-51.384,-178.272,5.883,148.532
C06065=1211.592,131.760,-51.364,-178.275,5.883,148.533
C06066=1211.597,131.511,-51.344,-178.277,5.882,148.533
C06067=1211.601,131.262,-51.324,-178.280,5.880,148.533
C06068=1211.607,131.012,-51.303,-178.282,5.879,148.534
C06069=1211.611,130.763,-51.283,-178.285,5.877,148.534
C06070=1211.615,130.514,-51.263,-178.288,5.877,148.535
C06071=1211.621,130.265,-51.243,-178.290,5.875,148.536
C06072=1211.625,130.016,-51.223,-178.293,5.874,148.536
C06073=1211.630,129.767,-51.203,-178.296,5.873,148.537
C06074=1211.634,129.518,-51.183,-178.298,5.872,148.537
C06075=1211.639,129.268,-51.163,-178.301,5.870,148.538
C06076=1211.644,129.019,-51.142,-178.303,5.869,148.538
C06077=1211.650,128.770,-51.123,-178.306,5.868,148.539
C06078=1211.654,128.521,-51.103,-178.308,5.867,148.539
C06079=1211.658,128.272,-51.082,-178.312,5.865,148.540
C06080=1211.663,128.022,-51.063,-178.314,5.865,148.540
C06081=1211.668,127.774,-51.042,-178.316,5.863,148.540
C06082=1211.673,127.525,-51.023,-178.319,5.862,148.541
C06083=1211.678,127.275,-51.003,-178.321,5.861,148.541
C06084=1211.682,127.026,-50.983,-178.324,5.860,148.542
C06085=1211.687,126.777,-50.963,-178.326,5.859,148.542
C06086=1211.691,126.528,-50.943,-178.330,5.857,148.543
C06087=1211.697,126.279,-50.924,-178.332,5.856,148.543
C06088=1211.701,126.030,-50.903,-178.335,5.855,148.544
C06089=1211.706,125.780,-50.884,-178.337,5.854,148.545
C06090=1211.710,125.531,-50.863,-178.340,5.852,148.545
C06091=1211.715,125.282,-50.843,-178.342,5.852,148.546
C06092=1211.720,125.033,-50.824,-178.345,5.850,148.546
C06093=1211.725,124.784,-50.804,-178.348,5.849,148.547
C06094=1211.730,124.534,-50.784,-178.350,5.848,148.547
C06095=1211.734,124.285,-50.765,-178.353,5.847,148.548
C06096=1211.739,124.037,-50.745,-178.355,5.846,148.548
C06097=1211.744,123.787,-50.725,-178.358,5.844,148.549
C06098=1211.749,123.537,-50.705,-178.360,5.843,148.549
C06099=1211.753,123.288,-50.685,-178.363,5.842,148.550
C06100=1211.759,123.040,-50.666,-178.366,5.841,148.550
C06101=1211.763,122.790,-50.646,-178.368,5.840,148.550
C06102=1211.768,122.541,-50.625,-178.371,5.839,148.551
C06103=1211.773,122.292,-50.606,-178.373,5.838,148.551
C06104=1211.778,122.043,-50.587,-178.376,5.836,148.552
C06105=1211.783,121.793,-50.567,-178.378,5.835,148.553
C06106=1211.787,121.544,-50.547,-178.381,5.834,148.553
C06107=1211.792,121.295,-50.527,-178.384,5.833,148.554
C06108=1211.797,121.046,-50.508,-178.386,5.832,148.554
C06109=1211.802,120.796,-50.488,-178.389,5.831,148.555
C06110=1211.806,120.548,-50.469,-178.391,5.830,148.555
C06111=1211.811,120.299,-50.449,-178.394,5.828,148.556
C06112=1211.816,120.049,-50.429,-178.397,5.828,148.556
C06113=1211.821,119.800,-50.410,-178.399,5.827,148.557
C06114=1211.826,119.551,-50.390,-178.402,5.825,148.557
C06115=1211.831,119.301,-50.371,-178.404,5.824,148.558
C06116=1211.836,119.053,-50.351,-178.407,5.823,148.558
C06117=1211.840,118.804,-50.332,-178.409,5.822,148.559
C06118=1211.844,118.554,-50.312,-178.413,5.820,148.559
C06119=1211.850,118.305,-50.293,-178.415,5.819,148.560
C06120=1211.854,118.056,-50.273,-178.417,5.819,148.560
C06121=1211.859,117.806,-50.253,-178.420,5.817,148.561
C06122=1211.865,117.557,-50.234,-178.423,5.816,148.561
C06123=1211.869,117.308,-50.215,-178.425,5.815,148.562
C06124=1211.874,117.059,-50.196,-178.428,5.814,148.562
C06125=1211.878,116.810,-50.175,-178.430,5.813,148.563
C06126=1211.883,116.560,-50.156,-178.433,5.812,148.564
C06127=1211.888,116.312,-50.136,-178.435,5.811,148.564
C06128=1211.892,116.062,-50.117,-178.438,5.810,148.565
C06129=1211.897,115.813,-50.098,-178.441,5.808,148.565
C06130=1211.902,115.564,-50.078,-178.443,5.808,148.566
C06131=1211.907,115.314,-50.059,-178.446,5.806,148.566
C06132=1211.912,115.066,-50.040,-178.449,5.805,148.567
C06133=1211.917,114.816,-50.020,-178.451,5.804,148.567
C06134=1211.922,114.567,-50.001,-178.454,5.803,148.568
C06135=1211.927,114.318,-49.981,-178.456,5.802,148.568
C06136=1211.931,114.068,-49.962,-178.459,5.801,148.569
C06137=1211.936,113.820,-49.943,-178.461,5.800,148.569
C06138=1211.941,113.570,-49.923,-178.464,5.799,148.570
C06139=1211.946,113.321,-49.905,-178.467,5.797,148.570
C06140=1211.950,113.071,-49.886,-178.469,5.797,148.571
C06141=1211.956,112.822,-49.866,-178.471,5.796,148.571
C06142=1211.960,112.573,-49.847,-178.475,5.794,148.572
C06143=1211.964,112.324,-49.828,-178.477,5.793,148.572
C06144=1211.970,112.075,-49.808,-178.480,5.792,148.573
C06145=1211.974,111.825,-49.789,-178.482,5.791,148.573
C06146=1211.979,111.577,-49.770,-178.485,5.790,148.574
C06147=1211.984,111.327,-49.750,-178.487,5.789,148.574
C06148=1211.989,111.078,-49.732,-178.490,5.788,148.575
C06149=1211.994,110.828,-49.713,-178.492,5.787,148.575
C06150=1211.999,110.579,-49.693,-178.495,5.786,148.576
C06151=1212.003,110.330,-49.674,-178.497,5.785,148.576
C06152=1212.008,110.081,-49.655,-178.500,5.784,148.577
C06153=1212.013,109.832,-49.635,-178.503,5.782,148.577
C06154=1212.018,109.583,-49.617,-178.505,5.782,148.578
C06155=1212.023,109.333,-49.598,-178.508,5.781,148.579
C06156=1212.027,109.084,-49.579,-178.511,5.779,148.579
C06157=1212.032,108.835,-49.559,-178.513,5.779,148.580
C06158=1212.037,108.586,-49.541,-178.516,5.777,148.580
C06159=1212.042,108.336,-49.522,-178.518,5.776,148.581
C06160=1212.047,108.087,-49.503,-178.521,5.775,148.581
C06161=1212.051,107.838,-49.483,-178.524,5.774,148.582
C06162=1212.057,107.569,-49.463,-178.526,5.773,148.583
C06163=1212.062,107.301,-49.442,-178.529,5.772,148.583
C06164=1212.067,107.033,-49.423,-178.532,5.771,148.584
C06165=1212.072,106.765,-49.402,-178.535,5.770,148.584
C06166=1212.077,106.515,-49.383,-178.537,5.769,148.585
C06167=1212.082,106.266,-49.365,-178.540,5.768,148.585
C06168=1212.087,106.016,-49.345,-178.542,5.766,148.586
C06169=1212.091,105.768,-49.326,-178.545,5.766,148.586
C06170=1212.096,105.518,-49.307,-178.548,5.765,148.587
C06171=1212.101,105.269,-49.289,-178.550,5.763,148.587
C06172=1212.106,105.019,-49.269,-178.553,5.763,148.588
C06173=1212.111,104.770,-49.251,-178.555,5.762,148.588
C06174=1212.116,104.521,-49.232,-178.558,5.760,148.589
C06175=1212.120,104.272,-49.213,-178.560,5.759,148.589
C06176=1212.126,104.023,-49.194,-178.563,5.759,148.590
C06177=1212.130,103.773,-49.175,-178.566,5.757,148.591
C06178=1212.135,103.524,-49.157,-178.568,5.757,148.591
C06179=1212.140,103.275,-49.138,-178.571,5.756,148.592
C06180=1212.144,103.025,-49.119,-178.573,5.755,148.592
C06181=1212.150,102.777,-49.100,-178.576,5.754,148.593
C06182=1212.154,102.527,-49.082,-178.578,5.753,148.593
C06183=1212.159,102.278,-49.062,-178.581,5.752,148.594
C06184=1212.164,102.029,-49.044,-178.584,5.750,148.594
C06185=1212.168,101.779,-49.025,-178.586,5.750,148.595
C06186=1212.174,101.530,-49.007,-178.589,5.749,148.596
C06187=1212.178,101.281,-48.988,-178.592,5.747,148.596
C06188=1212.183,101.031,-48.970,-178.594,5.747,148.597
C06189=1212.188,100.783,-48.951,-178.596,5.746,148.597
C06190=1212.192,100.533,-48.932,-178.599,5.744,148.598
C06191=1212.198,100.284,-48.913,-178.602,5.744,148.598
C06192=1212.203,100.035,-48.895,-178.604,5.743,148.599
C06193=1212.207,99.785,-48.877,-178.607,5.742,148.599
C06194=1212.212,99.536,-48.857,-178.610,5.740,148.600
C06195=1212.217,99.287,-48.839,-178.612,5.740,148.601
C06196=1212.221,99.038,-48.820,-178.614,5.739,148.601
C06197=1212.227,98.788,-48.802,-178.617,5.738,148.602
C06198=1212.232,98.539,-48.784,-178.620,5.737,148.602
C06199=1212.236,98.290,-48.765,-178.622,5.736,148.603
C06200=1212.241,98.040,-48.746,-178.625,5.735,148.603
C06201=1212.246,97.792,-48.727,-178.628,5.734,148.604
C06202=1212.251,97.542,-48.709,-178.630,5.733,148.604
C06203=1212.255,97.293,-48.691,-178.633,5.732,148.605
C06204=1212.261,97.044,-48.672,-178.635,5.731,148.605
C06205=1212.266,96.794,-48.654,-178.638,5.730,148.606
C06206=1212.270,96.545,-48.635,-178.640,5.729,148.606
C06207=1212.275,96.295,-48.617,-178.643,5.729,148.607
C06208=1212.280,96.047,-48.598,-178.646,5.727,148.608
C06209=1212.285,95.797,-48.580,-178.648,5.726,148.608
C06210=1212.289,95.548,-48.562,-178.651,5.726,148.609
C06211=1212.295,95.299,-48.543,-178.653,5.725,148.609
C06212=1212.300,95.049,-48.525,-178.656,5.723,148.610
C06213=1212.304,94.800,-48.506,-178.659,5.723,148.611
C06214=1212.309,94.550,-48.488,-178.661,5.722,148.611
C06215=1212.313,94.302,-48.470,-178.664,5.720,148.612
C06216=1212.319,94.052,-48.451,-178.667,5.720,148.612
C06217=1212.323,93.802,-48.433,-178.669,5.719,148.613
C06218=1212.328,93.553,-48.415,-178.671,5.718,148.613
C06219=1212.333,93.304,-48.397,-178.674,5.717,148.614
C06220=1212.338,93.056,-48.378,-178.677,5.716,148.614
C06221=1212.343,92.806,-48.360,-178.679,5.715,148.615
C06222=1212.348,92.556,-48.341,-178.681,5.714,148.615
C06223=1212.353,92.307,-48.323,-178.685,5.713,148.616
C06224=1212.358,92.058,-48.305,-178.687,5.712,148.616
C06225=1212.362,91.809,-48.287,-178.689,5.711,148.617
C06226=1212.367,91.559,-48.269,-178.692,5.711,148.618
C06227=1212.371,91.310,-48.250,-178.695,5.709,148.618
C06228=1212.377,91.061,-48.231,-178.697,5.709,148.619
C06229=1212.382,90.812,-48.213,-178.700,5.708,148.620
C06230=1212.387,90.562,-48.196,-178.702,5.707,148.620
C06231=1212.391,90.313,-48.177,-178.705,5.706,148.621
C06232=1212.396,90.063,-48.159,-178.708,5.705,148.621
C06233=1212.401,89.814,-48.141,-178.710,5.704,148.622
C06234=1212.406,89.565,-48.123,-178.713,5.704,148.622
C06235=1212.411,89.316,-48.105,-178.715,5.702,148.623
C06236=1212.416,89.067,-48.087,-178.718,5.701,148.623
C06237=1212.420,88.817,-48.069,-178.721,5.701,148.624
C06238=1212.425,88.568,-48.051,-178.723,5.700,148.624
C06239=1212.430,88.318,-48.033,-178.725,5.699,148.625
C06240=1212.436,88.069,-48.014,-178.729,5.698,148.626
C06241=1212.440,87.820,-47.996,-178.731,5.697,148.626
C06242=1212.445,87.571,-47.978,-178.733,5.696,148.627
C06243=1212.450,87.321,-47.960,-178.736,5.696,148.627
C06244=1212.455,87.072,-47.942,-178.739,5.694,148.628
C06245=1212.459,86.822,-47.924,-178.741,5.693,148.629
C06246=1212.464,86.573,-47.906,-178.743,5.692,148.629
C06247=1212.469,86.324,-47.888,-178.746,5.692,148.630
C06248=1212.474,86.075,-47.870,-178.749,5.691,148.630
C06249=1212.479,85.826,-47.852,-178.751,5.689,148.631
C06250=1212.484,85.576,-47.834,-178.754,5.689,148.631
C06251=1212.489,85.327,-47.816,-178.757,5.688,148.632
C06252=1212.494,85.077,-47.799,-178.759,5.687,148.632
C06253=1212.498,84.828,-47.781,-178.762,5.686,148.633
C06254=1212.503,84.578,-47.763,-178.765,5.685,148.634
C06255=1212.508,84.329,-47.745,-178.767,5.684,148.634
C06256=1212.512,84.080,-47.727,-178.769,5.684,148.635
C06257=1212.517,83.831,-47.709,-178.772,5.683,148.635
C06258=1212.522,83.582,-47.691,-178.775,5.681,148.636
C06259=1212.528,83.332,-47.674,-178.777,5.681,148.637
C06260=1212.532,83.083,-47.656,-178.780,5.680,148.637
C06261=1212.537,82.834,-47.638,-178.782,5.679,148.638
C06262=1212.542,82.585,-47.620,-178.785,5.679,148.638
C06263=1212.547,82.336,-47.602,-178.788,5.677,148.639
C06264=1212.552,82.086,-47.585,-178.790,5.676,148.639
C06265=1212.557,81.837,-47.567,-178.793,5.676,148.640
C06266=1212.562,81.568,-47.547,-178.795,5.675,148.641
C06267=1212.568,81.299,-47.529,-178.798,5.674,148.641
C06268=1212.573,81.031,-47.509,-178.801,5.673,148.642
C06269=1212.578,80.763,-47.490,-178.804,5.673,148.643
C06270=1212.583,80.513,-47.473,-178.806,5.671,148.643
C06271=1212.587,80.264,-47.455,-178.809,5.670,148.644
C06272=1212.592,80.015,-47.437,-178.812,5.670,148.644
C06273=1212.597,79.766,-47.419,-178.814,5.669,148.645
C06274=1212.602,79.516,-47.402,-178.816,5.668,148.645
C06275=1212.607,79.267,-47.384,-178.819,5.668,148.646
C06276=1212.612,79.018,-47.366,-178.822,5.666,148.646
C06277=1212.617,78.768,-47.349,-178.824,5.665,148.647
C06278=1212.622,78.519,-47.331,-178.827,5.665,148.648
C06279=1212.626,78.270,-47.314,-178.829,5.664,148.648
C06280=1212.632,78.020,-47.296,-178.832,5.663,148.649
C06281=1212.637,77.771,-47.278,-178.835,5.662,148.650
C06282=1212.641,77.522,-47.262,-178.837,5.661,148.650
C06283=1212.646,77.272,-47.244,-178.840,5.661,148.651
C06284=1212.651,77.023,-47.226,-178.842,5.660,148.651
C06285=1212.656,76.773,-47.208,-178.844,5.659,148.652
C06286=1212.661,76.524,-47.190,-178.847,5.658,148.652
C06287=1212.666,76.275,-47.174,-178.850,5.657,148.653
C06288=1212.670,76.026,-47.156,-178.853,5.656,148.654
C06289=1212.676,75.776,-47.138,-178.855,5.656,148.654
C06290=1212.680,75.527,-47.121,-178.858,5.655,148.655
C06291=1212.685,75.278,-47.103,-178.860,5.654,148.655
C06292=1212.690,75.028,-47.086,-178.862,5.653,148.656
C06293=1212.695,74.779,-47.068,-178.865,5.653,148.657
C06294=1212.700,74.530,-47.052,-178.868,5.652,148.657
C06295=1212.705,74.281,-47.034,-178.870,5.651,148.658
C06296=1212.710,74.031,-47.016,-178.873,5.650,148.658
C06297=1212.714,73.782,-46.999,-178.876,5.649,148.659
C06298=1212.719,73.532,-46.982,-178.878,5.649,148.660
C06299=1212.725,73.283,-46.964,-178.880,5.648,148.660
C06300=1212.730,73.033,-46.946,-178.884,5.647,148.661
C06301=1212.734,72.784,-46.930,-178.886,5.646,148.661
C06302=1212.739,72.535,-46.912,-178.888,5.645,148.662
C06303=1212.744,72.285,-46.895,-178.891,5.645,148.662
C06304=1212.748,72.036,-46.877,-178.894,5.644,148.663
C06305=1212.754,71.787,-46.860,-178.896,5.643,148.664
C06306=1212.759,71.537,-46.844,-178.898,5.642,148.664
C06307=1212.764,71.288,-46.826,-178.902,5.641,148.665
C06308=1212.769,71.038,-46.808,-178.904,5.640,148.665
C06309=1212.773,70.790,-46.791,-178.906,5.640,148.666
C06310=1212.778,70.540,-46.774,-178.909,5.639,148.667
C06311=1212.783,70.290,-46.756,-178.912,5.638,148.667
C06312=1212.788,70.041,-46.739,-178.914,5.638,148.668
C06313=1212.793,69.792,-46.722,-178.916,5.637,148.668
C06314=1212.798,69.543,-46.705,-178.919,5.636,148.669
C06315=1212.803,69.293,-46.687,-178.922,5.635,148.670
C06316=1212.808,69.044,-46.670,-178.924,5.634,148.670
C06317=1212.813,68.794,-46.654,-178.927,5.634,148.671
C06318=1212.817,68.545,-46.636,-178.930,5.633,148.671
C06319=1212.822,68.295,-46.619,-178.932,5.632,148.672
C06320=1212.828,68.046,-46.602,-178.934,5.631,148.672
C06321=1212.832,67.797,-46.585,-178.937,5.631,148.673
C06322=1212.837,67.548,-46.567,-178.940,5.630,148.674
C06323=1212.842,67.298,-46.551,-178.943,5.629,148.674
C06324=1212.847,67.048,-46.533,-178.945,5.628,148.675
C06325=1212.852,66.800,-46.517,-178.948,5.627,148.676
C06326=1212.857,66.550,-46.499,-178.950,5.627,148.676
C06327=1212.861,66.301,-46.482,-178.952,5.626,148.677
C06328=1212.867,66.051,-46.465,-178.955,5.625,148.677
C06329=1212.871,65.802,-46.449,-178.958,5.625,148.678
C06330=1212.877,65.553,-46.431,-178.960,5.624,148.679
C06331=1212.881,65.304,-46.414,-178.962,5.623,148.679
C06332=1212.886,65.054,-46.397,-178.966,5.622,148.680
C06333=1212.891,64.804,-46.380,-178.968,5.621,148.680
C06334=1212.896,64.555,-46.363,-178.971,5.621,148.681
C06335=1212.901,64.306,-46.347,-178.973,5.620,148.681
C06336=1212.906,64.056,-46.329,-178.976,5.619,148.682
C06337=1212.910,63.807,-46.312,-178.978,5.619,148.683
C06338=1212.916,63.557,-46.295,-178.981,5.618,148.683
C06339=1212.921,63.309,-46.279,-178.983,5.617,148.684
C06340=1212.925,63.059,-46.262,-178.986,5.617,148.685
C06341=1212.930,62.809,-46.245,-178.988,5.616,148.685
C06342=1212.935,62.560,-46.228,-178.991,5.616,148.686
C06343=1212.941,62.311,-46.211,-178.994,5.614,148.686
C06344=1212.945,62.061,-46.194,-178.996,5.613,148.687
C06345=1212.950,61.812,-46.177,-178.999,5.613,148.688
C06346=1212.955,61.562,-46.160,-179.002,5.612,148.688
C06347=1212.960,61.313,-46.144,-179.004,5.611,148.689
C06348=1212.965,61.063,-46.127,-179.006,5.611,148.689
C06349=1212.969,60.815,-46.109,-179.009,5.610,148.690
C06350=1212.974,60.566,-46.093,-179.012,5.610,148.691
C06351=1212.980,60.316,-46.076,-179.014,5.609,148.691
C06352=1212.984,60.067,-46.059,-179.016,5.608,148.692
C06353=1212.989,59.817,-46.042,-179.019,5.608,148.693
C06354=1212.995,59.567,-46.026,-179.022,5.607,148.693
C06355=1212.999,59.318,-46.010,-179.024,5.605,148.694
C06356=1213.004,59.068,-45.992,-179.027,5.605,148.694
C06357=1213.009,58.819,-45.976,-179.030,5.604,148.695
C06358=1213.014,58.570,-45.959,-179.032,5.604,148.696
C06359=1213.019,58.320,-45.942,-179.034,5.603,148.696
C06360=1213.024,58.071,-45.926,-179.037,5.602,148.697
C06361=1213.029,57.822,-45.909,-179.040,5.602,148.697
C06362=1213.033,57.572,-45.893,-179.042,5.601,148.698
C06363=1213.039,57.323,-45.876,-179.045,5.600,148.699
C06364=1213.044,57.074,-45.859,-179.047,5.600,148.699
C06365=1213.048,56.824,-45.842,-179.050,5.599,148.700
C06366=1213.054,56.575,-45.825,-179.052,5.598,148.700
C06367=1213.059,56.325,-45.809,-179.055,5.598,148.701
C06368=1213.063,56.075,-45.793,-179.057,5.597,148.702
C06369=1213.068,55.827,-45.777,-179.060,5.596,148.702
C06370=1213.074,55.558,-45.758,-179.063,5.595,148.703
C06371=1213.079,55.290,-45.740,-179.066,5.595,148.704
C06372=1213.084,55.022,-45.723,-179.068,5.594,148.704
C06373=1213.090,54.753,-45.704,-179.071,5.593,148.705
C06374=1213.095,54.504,-45.688,-179.074,5.593,148.706
C06375=1213.100,54.254,-45.672,-179.076,5.592,148.706
C06376=1213.104,54.004,-45.655,-179.078,5.591,148.707
C06377=1213.109,53.755,-45.639,-179.081,5.591,148.707
C06378=1213.114,53.506,-45.622,-179.084,5.589,148.708
C06379=1213.119,53.257,-45.606,-179.087,5.589,148.709
C06380=1213.124,53.007,-45.590,-179.089,5.588,148.709
C06381=1213.129,52.757,-45.573,-179.092,5.587,148.710
C06382=1213.134,52.509,-45.557,-179.094,5.587,148.710
C06383=1213.139,52.258,-45.540,-179.097,5.586,148.711
C06384=1213.144,52.009,-45.524,-179.100,5.586,148.712
C06385=1213.149,51.760,-45.507,-179.102,5.585,148.712
C06386=1213.153,51.510,-45.490,-179.104,5.584,148.713
C06387=1213.159,51.261,-45.475,-179.107,5.584,148.714
C06388=1213.163,51.011,-45.458,-179.110,5.583,148.714
C06389=1213.168,50.763,-45.442,-179.112,5.583,148.715
C06390=1213.174,50.512,-45.425,-179.114,5.582,148.715
C06391=1213.179,50.264,-45.409,-179.117,5.581,148.716
C06392=1213.183,50.014,-45.392,-179.120,5.581,148.717
C06393=1213.189,49.765,-45.377,-179.122,5.580,148.717
C06394=1213.193,49.515,-45.360,-179.125,5.580,148.718
C06395=1213.198,49.266,-45.343,-179.127,5.579,148.718
C06396=1213.203,49.016,-45.328,-179.130,5.578,148.719
C06397=1213.208,48.767,-45.311,-179.132,5.578,148.720
C06398=1213.213,48.517,-45.296,-179.135,5.577,148.720
C06399=1213.218,48.268,-45.279,-179.138,5.576,148.721
C06400=1213.223,48.019,-45.262,-179.140,5.576,148.722
C06401=1213.228,47.769,-45.246,-179.142,5.575,148.722
C06402=1213.233,47.520,-45.230,-179.145,5.574,148.723
C06403=1213.238,47.270,-45.214,-179.148,5.574,148.724
C06404=1213.243,47.021,-45.198,-179.150,5.573,148.724
C06405=1213.248,46.771,-45.182,-179.152,5.572,148.725
C06406=1213.253,46.522,-45.165,-179.155,5.572,148.725
C06407=1213.258,46.272,-45.149,-179.158,5.571,148.726
C06408=1213.263,46.023,-45.133,-179.160,5.571,148.727
C06409=1213.268,45.773,-45.117,-179.163,5.570,148.727
C06410=1213.273,45.524,-45.101,-179.166,5.570,148.728
C06411=1213.277,45.274,-45.085,-179.168,5.569,148.729
C06412=1213.283,45.025,-45.068,-179.170,5.568,148.729
C06413=1213.287,44.775,-45.053,-179.173,5.568,148.730
C06414=1213.292,44.527,-45.036,-179.176,5.567,148.731
C06415=1213.298,44.277,-45.021,-179.178,5.567,148.731
C06416=1213.302,44.028,-45.004,-179.181,5.566,148.732
C06417=1213.308,43.778,-44.988,-179.183,5.565,148.732
C06418=1213.312,43.529,-44.972,-179.186,5.565,148.733
C06419=1213.318,43.279,-44.956,-179.188,5.564,148.734
C06420=1213.322,43.030,-44.939,-179.191,5.564,148.734
C06421=1213.327,42.781,-44.924,-179.193,5.563,148.735
C06422=1213.332,42.530,-44.908,-179.196,5.562,148.735
C06423=1213.337,42.282,-44.892,-179.198,5.562,148.736
C06424=1213.342,42.033,-44.877,-179.201,5.561,148.737
C06425=1213.347,41.782,-44.861,-179.204,5.560,148.737
C06426=1213.352,41.534,-44.844,-179.206,5.560,148.738
C06427=1213.357,41.284,-44.828,-179.209,5.559,148.739
C06428=1213.362,41.035,-44.812,-179.211,5.558,148.739
C06429=1213.367,40.785,-44.797,-179.214,5.558,148.740
C06430=1213.372,40.535,-44.781,-179.216,5.557,148.741
C06431=1213.377,40.286,-44.764,-179.219,5.557,148.741
C06432=1213.382,40.036,-44.748,-179.221,5.556,148.742
C06433=1213.387,39.787,-44.733,-179.224,5.555,148.742
C06434=1213.392,39.538,-44.718,-179.227,5.555,148.743
C06435=1213.396,39.288,-44.701,-179.229,5.554,148.744
C06436=1213.402,39.039,-44.685,-179.232,5.554,148.744
C06437=1213.406,38.789,-44.670,-179.234,5.553,148.745
C06438=1213.411,38.540,-44.653,-179.237,5.552,148.746
C06439=1213.417,38.291,-44.638,-179.239,5.552,148.746
C06440=1213.422,38.041,-44.622,-179.242,5.551,148.747
C06441=1213.426,37.792,-44.607,-179.245,5.551,148.748
C06442=1213.432,37.542,-44.591,-179.247,5.550,148.748
C06443=1213.436,37.293,-44.574,-179.250,5.550,148.749
C06444=1213.442,37.043,-44.559,-179.252,5.549,148.749
C06445=1213.447,36.794,-44.543,-179.255,5.548,148.750
C06446=1213.451,36.544,-44.528,-179.257,5.548,148.751
C06447=1213.456,36.295,-44.512,-179.260,5.547,148.751
C06448=1213.461,36.046,-44.496,-179.263,5.547,148.752
C06449=1213.466,35.796,-44.480,-179.265,5.546,148.753
C06450=1213.472,35.546,-44.464,-179.267,5.545,148.753
C06451=1213.476,35.297,-44.449,-179.270,5.545,148.754
C06452=1213.481,35.047,-44.434,-179.272,5.545,148.755
C06453=1213.486,34.798,-44.418,-179.275,5.544,148.755
C06454=1213.491,34.549,-44.402,-179.277,5.544,148.756
C06455=1213.496,34.299,-44.386,-179.280,5.543,148.757
C06456=1213.501,34.050,-44.371,-179.283,5.543,148.757
C06457=1213.506,33.800,-44.355,-179.285,5.542,148.758
C06458=1213.512,33.551,-44.340,-179.287,5.541,148.758
C06459=1213.516,33.301,-44.324,-179.290,5.541,148.759
C06460=1213.521,33.052,-44.309,-179.293,5.540,148.760
C06461=1213.527,32.802,-44.293,-179.295,5.540,148.760
C06462=1213.531,32.553,-44.278,-179.298,5.539,148.761
C06463=1213.536,32.303,-44.262,-179.300,5.538,148.762
C06464=1213.541,32.054,-44.246,-179.303,5.538,148.762
C06465=1213.546,31.805,-44.231,-179.305,5.537,148.763
C06466=1213.550,31.555,-44.215,-179.308,5.537,148.764
C06467=1213.556,31.306,-44.199,-179.311,5.536,148.764
C06468=1213.561,31.056,-44.184,-179.313,5.536,148.765
C06469=1213.566,30.807,-44.169,-179.316,5.535,148.766
C06470=1213.571,30.557,-44.153,-179.318,5.535,148.766
C06471=1213.575,30.308,-44.138,-179.320,5.534,148.767
C06472=1213.581,30.059,-44.122,-179.323,5.534,148.767
C06473=1213.586,29.809,-44.106,-179.326,5.533,148.768
C06474=1213.591,29.541,-44.091,-179.328,5.533,148.769
C06475=1213.596,29.271,-44.073,-179.331,5.532,148.769
C06476=1213.602,29.002,-44.057,-179.333,5.532,148.770
C06477=1213.607,28.734,-44.041,-179.337,5.530,148.771
C06478=1213.612,28.485,-44.025,-179.339,5.531,148.771
C06479=1213.618,28.235,-44.009,-179.341,5.530,148.772
C06480=1213.622,27.986,-43.994,-179.344,5.530,148.773
C06481=1213.627,27.736,-43.979,-179.347,5.529,148.773
C06482=1213.632,27.487,-43.964,-179.349,5.529,148.774
C06483=1213.637,27.237,-43.949,-179.351,5.528,148.775
C06484=1213.643,26.988,-43.933,-179.354,5.527,148.775
C06485=1213.647,26.738,-43.918,-179.357,5.527,148.776
C06486=1213.652,26.488,-43.902,-179.359,5.526,148.777
C06487=1213.657,26.239,-43.887,-179.362,5.526,148.777
C06488=1213.662,25.990,-43.872,-179.365,5.525,148.778
C06489=1213.667,25.741,-43.857,-179.367,5.524,148.779
C06490=1213.673,25.491,-43.842,-179.370,5.524,148.779
C06491=1213.678,25.241,-43.826,-179.372,5.524,148.780
C06492=1213.682,24.992,-43.811,-179.374,5.523,148.780
C06493=1213.687,24.742,-43.795,-179.377,5.523,148.781
C06494=1213.692,24.493,-43.780,-179.380,5.522,148.782
C06495=1213.697,24.244,-43.765,-179.382,5.522,148.783
C06496=1213.702,23.994,-43.750,-179.385,5.521,148.783
C06497=1213.708,23.745,-43.735,-179.387,5.521,148.784
C06498=1213.712,23.495,-43.720,-179.390,5.520,148.784
C06499=1213.717,23.245,-43.704,-179.392,5.519,148.785
C06500=1213.722,22.996,-43.689,-179.395,5.519,148.786
C06501=1213.728,22.746,-43.674,-179.397,5.519,148.786
C06502=1213.732,22.497,-43.659,-179.400,5.518,148.787
C06503=1213.737,22.248,-43.644,-179.402,5.518,148.788
C06504=1213.743,21.998,-43.629,-179.405,5.517,148.788
C06505=1213.747,21.749,-43.614,-179.408,5.517,148.789
C06506=1213.753,21.500,-43.598,-179.410,5.516,148.790
C06507=1213.757,21.249,-43.584,-179.412,5.515,148.790
C06508=1213.762,21.000,-43.568,-179.415,5.515,148.791
C06509=1213.767,20.751,-43.553,-179.418,5.514,148.792
C06510=1213.773,20.501,-43.538,-179.420,5.515,148.792
C06511=1213.777,20.252,-43.523,-179.422,5.514,148.793
C06512=1213.782,20.002,-43.508,-179.425,5.514,148.794
C06513=1213.788,19.752,-43.494,-179.428,5.513,148.794
C06514=1213.792,19.503,-43.479,-179.430,5.512,148.795
C06515=1213.798,19.254,-43.463,-179.432,5.512,148.795
C06516=1213.803,19.004,-43.449,-179.435,5.511,148.796
C06517=1213.807,18.755,-43.434,-179.438,5.511,148.797
C06518=1213.812,18.504,-43.418,-179.440,5.510,148.798
C06519=1213.817,18.255,-43.403,-179.442,5.510,148.798
C06520=1213.822,18.006,-43.388,-179.445,5.510,148.799
C06521=1213.827,17.756,-43.374,-179.448,5.509,148.800
C06522=1213.832,17.507,-43.359,-179.450,5.509,148.800
C06523=1213.838,17.257,-43.344,-179.453,5.508,148.801
C06524=1213.842,17.008,-43.329,-179.455,5.507,148.801
C06525=1213.847,16.758,-43.314,-179.458,5.507,148.802
C06526=1213.853,16.509,-43.299,-179.461,5.506,148.803
C06527=1213.858,16.259,-43.285,-179.463,5.507,148.803
C06528=1213.862,16.010,-43.270,-179.465,5.506,148.804
C06529=1213.868,15.761,-43.254,-179.468,5.506,148.805
C06530=1213.873,15.511,-43.240,-179.471,5.505,148.805
C06531=1213.877,15.262,-43.225,-179.473,5.504,148.806
C06532=1213.883,15.012,-43.210,-179.475,5.504,148.807
C06533=1213.888,14.762,-43.196,-179.478,5.503,148.807
C06534=1213.893,14.513,-43.181,-179.480,5.503,148.808
C06535=1213.898,14.263,-43.166,-179.483,5.503,148.809
C06536=1213.903,14.014,-43.151,-179.485,5.502,148.809
C06537=1213.908,13.764,-43.136,-179.488,5.502,148.810
C06538=1213.913,13.515,-43.121,-179.491,5.501,148.811
C06539=1213.918,13.265,-43.107,-179.493,5.501,148.811
C06540=1213.923,13.016,-43.092,-179.496,5.500,148.812
C06541=1213.928,12.766,-43.077,-179.498,5.499,148.813
C06542=1213.933,12.517,-43.063,-179.500,5.500,148.813
C06543=1213.937,12.267,-43.048,-179.503,5.499,148.814
C06544=1213.943,12.017,-43.033,-179.505,5.499,148.815
C06545=1213.948,11.768,-43.018,-179.508,5.498,148.815
C06546=1213.953,11.519,-43.004,-179.511,5.498,148.816
C06547=1213.958,11.269,-42.990,-179.513,5.497,148.817
C06548=1213.963,11.020,-42.974,-179.516,5.497,148.817
C06549=1213.968,10.770,-42.960,-179.518,5.497,148.818
C06550=1213.973,10.520,-42.945,-179.520,5.496,148.818
C06551=1213.978,10.271,-42.930,-179.523,5.496,148.819
C06552=1213.983,10.022,-42.917,-179.526,5.495,148.820
C06553=1213.989,9.772,-42.902,-179.528,5.495,148.821
C06554=1213.994,9.523,-42.887,-179.531,5.494,148.821
C06555=1213.999,9.273,-42.872,-179.533,5.494,148.822
C06556=1214.003,9.023,-42.858,-179.536,5.494,148.823
C06557=1214.008,8.774,-42.843,-179.538,5.493,148.823
C06558=1214.013,8.525,-42.829,-179.541,5.493,148.824
C06559=1214.019,8.275,-42.814,-179.544,5.492,148.825
C06560=1214.024,8.025,-42.800,-179.546,5.491,148.825
C06561=1214.028,7.776,-42.785,-179.548,5.492,148.826
C06562=1214.033,7.526,-42.770,-179.550,5.491,148.826
C06563=1214.038,7.276,-42.756,-179.553,5.491,148.827
C06564=1214.044,7.027,-42.742,-179.556,5.490,148.828
C06565=1214.049,6.778,-42.727,-179.558,5.490,148.829
C06566=1214.053,6.529,-42.713,-179.561,5.489,148.829
C06567=1214.058,6.279,-42.699,-179.563,5.489,148.830
C06568=1214.064,6.029,-42.684,-179.566,5.489,148.831
C06569=1214.069,5.779,-42.670,-179.568,5.488,148.831
C06570=1214.074,5.530,-42.655,-179.571,5.488,148.832
C06571=1214.079,5.280,-42.640,-179.573,5.487,148.832
C06572=1214.084,5.031,-42.626,-179.575,5.487,148.833
C06573=1214.089,4.782,-42.612,-179.578,5.487,148.834
C06574=1214.094,4.532,-42.598,-179.581,5.486,148.834
C06575=1214.099,4.282,-42.584,-179.583,5.486,148.835
C06576=1214.104,4.033,-42.569,-179.586,5.485,148.836
C06577=1214.109,3.783,-42.554,-179.589,5.485,148.837
C06578=1214.114,3.514,-42.539,-179.591,5.484,148.837
C06579=1214.119,3.245,-42.524,-179.593,5.484,148.838
C06580=1214.126,2.976,-42.508,-179.596,5.484,148.839
C06581=1214.131,2.707,-42.493,-179.599,5.483,148.839
C06582=1214.136,2.458,-42.478,-179.601,5.483,148.840
C06583=1214.141,2.208,-42.464,-179.604,5.482,148.841
C06584=1214.146,1.958,-42.450,-179.607,5.482,148.841
C06585=1214.151,1.709,-42.436,-179.609,5.481,148.842
C06586=1214.157,1.460,-42.422,-179.611,5.482,148.843
C06587=1214.161,1.210,-42.407,-179.614,5.481,148.843
C06588=1214.166,0.960,-42.393,-179.617,5.481,148.844
C06589=1214.171,0.710,-42.379,-179.619,5.480,148.845
C06590=1214.176,0.461,-42.364,-179.622,5.480,148.845
C06591=1214.182,0.212,-42.350,-179.624,5.480,148.846
C06592=1214.187,-0.037,-42.336,-179.626,5.479,148.847
C06593=1214.192,-0.287,-42.321,-179.629,5.479,148.847
C06594=1214.196,-0.537,-42.307,-179.631,5.478,148.848
C06595=1214.201,-0.785,-42.294,-179.634,5.478,148.849
C06596=1214.207,-1.036,-42.280,-179.636,5.478,148.849
C06597=1214.211,-1.286,-42.266,-179.639,5.477,148.850
C06598=1214.216,-1.535,-42.252,-179.642,5.477,148.851
C06599=1214.221,-1.785,-42.237,-179.644,5.476,148.851
C06600=1214.227,-2.034,-42.223,-179.647,5.476,148.852
C06601=1214.232,-2.284,-42.209,-179.649,5.476,148.853
C06602=1214.237,-2.533,-42.195,-179.652,5.476,148.854
C06603=1214.242,-2.783,-42.181,-179.654,5.475,148.854
C06604=1214.247,-3.032,-42.167,-179.656,5.474,148.855
C06605=1214.252,-3.282,-42.152,-179.659,5.474,148.855
C06606=1214.257,-3.532,-42.138,-179.661,5.474,148.856
C06607=1214.262,-3.781,-42.124,-179.664,5.474,148.857
C06608=1214.267,-4.030,-42.111,-179.666,5.473,148.857
C06609=1214.272,-4.280,-42.097,-179.669,5.473,148.858
C06610=1214.277,-4.530,-42.083,-179.672,5.472,148.859
C06611=1214.283,-4.779,-42.069,-179.674,5.472,148.860
C06612=1214.288,-5.029,-42.055,-179.676,5.472,148.860
C06613=1214.293,-5.278,-42.040,-179.679,5.471,148.861
C06614=1214.297,-5.528,-42.027,-179.682,5.471,148.862
C06615=1214.303,-5.777,-42.013,-179.684,5.471,148.862
C06616=1214.308,-6.027,-41.999,-179.686,5.471,148.863
C06617=1214.313,-6.277,-41.985,-179.689,5.470,148.863
C06618=1214.318,-6.526,-41.971,-179.691,5.469,148.864
C06619=1214.323,-6.775,-41.957,-179.694,5.469,148.865
C06620=1214.327,-7.025,-41.943,-179.696,5.469,148.866
C06621=1214.333,-7.275,-41.930,-179.699,5.469,148.866
C06622=1214.338,-7.524,-41.915,-179.701,5.468,148.867
C06623=1214.343,-7.774,-41.901,-179.704,5.468,148.868
C06624=1214.347,-8.023,-41.888,-179.706,5.468,148.868
C06625=1214.353,-8.273,-41.874,-179.709,5.467,148.869
C06626=1214.358,-8.523,-41.860,-179.711,5.467,148.870
C06627=1214.363,-8.772,-41.846,-179.714,5.466,148.870
C06628=1214.368,-9.021,-41.832,-179.716,5.467,148.871
C06629=1214.373,-9.271,-41.819,-179.719,5.466,148.872
C06630=1214.379,-9.520,-41.805,-179.721,5.465,148.872
C06631=1214.384,-9.770,-41.791,-179.724,5.465,148.873
C06632=1214.388,-10.020,-41.777,-179.726,5.464,148.874
C06633=1214.394,-10.269,-41.764,-179.728,5.465,148.874
C06634=1214.399,-10.519,-41.750,-179.731,5.464,148.875
C06635=1214.404,-10.769,-41.735,-179.734,5.464,148.876
C06636=1214.409,-11.018,-41.723,-179.736,5.463,148.876
C06637=1214.414,-11.268,-41.708,-179.738,5.463,148.877
C06638=1214.419,-11.517,-41.694,-179.741,5.463,148.878
C06639=1214.424,-11.767,-41.682,-179.744,5.462,148.878
C06640=1214.429,-12.016,-41.667,-179.746,5.462,148.879
C06641=1214.435,-12.266,-41.654,-179.748,5.462,148.880
C06642=1214.440,-12.516,-41.640,-179.751,5.462,148.880
C06643=1214.444,-12.765,-41.626,-179.754,5.461,148.881
C06644=1214.450,-13.015,-41.613,-179.756,5.460,148.882
C06645=1214.455,-13.265,-41.599,-179.758,5.461,148.882
C06646=1214.460,-13.514,-41.586,-179.761,5.460,148.883
C06647=1214.465,-13.764,-41.572,-179.763,5.460,148.884
C06648=1214.470,-14.013,-41.557,-179.766,5.459,148.884
C06649=1214.475,-14.263,-41.545,-179.768,5.460,148.885
C06650=1214.480,-14.512,-41.531,-179.771,5.459,148.886
C06651=1214.485,-14.762,-41.518,-179.773,5.459,148.887
C06652=1214.490,-15.011,-41.504,-179.776,5.458,148.887
C06653=1214.495,-15.262,-41.490,-179.778,5.458,148.888
C06654=1214.500,-15.510,-41.477,-179.781,5.458,148.889
C06655=1214.505,-15.761,-41.463,-179.783,5.457,148.889
C06656=1214.511,-16.010,-41.449,-179.786,5.457,148.890
C06657=1214.515,-16.260,-41.436,-179.788,5.457,148.891
C06658=1214.521,-16.509,-41.422,-179.791,5.457,148.891
C06659=1214.525,-16.759,-41.410,-179.793,5.456,148.892
C06660=1214.531,-17.008,-41.396,-179.795,5.456,148.893
C06661=1214.536,-17.258,-41.382,-179.798,5.456,148.893
C06662=1214.541,-17.507,-41.369,-179.800,5.455,148.894
C06663=1214.546,-17.757,-41.355,-179.803,5.455,148.895
C06664=1214.551,-18.006,-41.341,-179.805,5.455,148.895
C06665=1214.556,-18.256,-41.328,-179.808,5.454,148.896
C06666=1214.561,-18.506,-41.315,-179.810,5.454,148.897
C06667=1214.566,-18.755,-41.301,-179.813,5.454,148.897
C06668=1214.571,-19.005,-41.288,-179.815,5.454,148.898
C06669=1214.577,-19.254,-41.275,-179.818,5.453,148.899
C06670=1214.582,-19.505,-41.261,-179.820,5.453,148.899
C06671=1214.587,-19.753,-41.248,-179.823,5.452,148.900
C06672=1214.592,-20.004,-41.234,-179.825,5.453,148.901
C06673=1214.597,-20.253,-41.221,-179.828,5.452,148.902
C06674=1214.602,-20.503,-41.207,-179.830,5.451,148.902
C06675=1214.607,-20.752,-41.195,-179.832,5.452,148.903
C06676=1214.612,-21.002,-41.180,-179.835,5.451,148.903
C06677=1214.617,-21.251,-41.168,-179.837,5.451,148.904
C06678=1214.622,-21.501,-41.154,-179.840,5.450,148.905
C06679=1214.627,-21.750,-41.141,-179.842,5.450,148.905
C06680=1214.633,-22.000,-41.128,-179.845,5.450,148.906
C06681=1214.638,-22.250,-41.115,-179.847,5.449,148.907
C06682=1214.643,-22.519,-41.100,-179.850,5.449,148.908
C06683=1214.649,-22.788,-41.086,-179.852,5.449,148.908
C06684=1214.654,-23.057,-41.071,-179.855,5.449,148.909
C06685=1214.660,-23.327,-41.057,-179.858,5.449,148.910
C06686=1214.665,-23.577,-41.045,-179.861,5.448,148.911
C06687=1214.670,-23.827,-41.030,-179.863,5.448,148.911
C06688=1214.675,-24.076,-41.018,-179.865,5.448,148.912
C06689=1214.680,-24.326,-41.005,-179.868,5.447,148.912
C06690=1214.685,-24.575,-40.991,-179.870,5.447,148.913
C06691=1214.690,-24.824,-40.978,-179.872,5.447,148.914
C06692=1214.696,-25.074,-40.965,-179.875,5.447,148.915
C06693=1214.701,-25.324,-40.952,-179.878,5.446,148.915
C06694=1214.705,-25.574,-40.939,-179.880,5.446,148.916
C06695=1214.711,-25.823,-40.925,-179.882,5.446,148.917
C06696=1214.715,-26.073,-40.912,-179.885,5.445,148.917
C06697=1214.721,-26.322,-40.899,-179.888,5.445,148.918
C06698=1214.726,-26.572,-40.886,-179.890,5.445,148.919
C06699=1214.731,-26.822,-40.873,-179.892,5.445,148.919
C06700=1214.736,-27.071,-40.859,-179.895,5.444,148.920
C06701=1214.741,-27.321,-40.847,-179.897,5.445,148.921
C06702=1214.746,-27.570,-40.834,-179.900,5.444,148.922
C06703=1214.752,-27.820,-40.821,-179.903,5.444,148.922
C06704=1214.756,-28.070,-40.808,-179.905,5.444,148.923
C06705=1214.762,-28.319,-40.795,-179.907,5.443,148.923
C06706=1214.767,-28.569,-40.782,-179.909,5.443,148.924
C06707=1214.772,-28.818,-40.768,-179.912,5.442,148.925
C06708=1214.777,-29.068,-40.755,-179.914,5.442,148.925
C06709=1214.782,-29.318,-40.742,-179.917,5.442,148.926
C06710=1214.787,-29.567,-40.729,-179.919,5.441,148.927
C06711=1214.792,-29.816,-40.717,-179.922,5.442,148.928
C06712=1214.797,-30.067,-40.703,-179.924,5.441,148.928
C06713=1214.803,-30.316,-40.691,-179.927,5.441,148.929
C06714=1214.808,-30.565,-40.678,-179.929,5.441,148.930
C06715=1214.813,-30.816,-40.665,-179.932,5.441,148.930
C06716=1214.818,-31.065,-40.652,-179.934,5.440,148.931
C06717=1214.823,-31.314,-40.639,-179.936,5.441,148.932
C06718=1214.828,-31.564,-40.626,-179.939,5.440,148.932
C06719=1214.834,-31.814,-40.613,-179.942,5.440,148.933
C06720=1214.838,-32.063,-40.600,-179.944,5.440,148.934
C06721=1214.843,-32.313,-40.587,-179.946,5.439,148.935
C06722=1214.849,-32.562,-40.574,-179.949,5.439,148.935
C06723=1214.854,-32.812,-40.561,-179.951,5.438,148.936
C06724=1214.858,-33.062,-40.548,-179.953,5.438,148.936
C06725=1214.864,-33.311,-40.536,-179.956,5.438,148.937
C06726=1214.869,-33.561,-40.524,-179.959,5.437,148.938
C06727=1214.874,-33.811,-40.510,-179.961,5.438,148.938
C06728=1214.879,-34.061,-40.498,-179.963,5.437,148.939
C06729=1214.884,-34.310,-40.485,-179.966,5.437,148.940
C06730=1214.889,-34.560,-40.472,-179.968,5.437,148.941
C06731=1214.895,-34.810,-40.459,-179.971,5.437,148.941
C06732=1214.900,-35.059,-40.446,-179.974,5.436,148.942
C06733=1214.905,-35.308,-40.434,-179.976,5.436,148.943
C06734=1214.910,-35.558,-40.421,-179.978,5.436,148.943
C06735=1214.915,-35.808,-40.408,-179.981,5.436,148.944
C06736=1214.921,-36.057,-40.395,-179.983,5.436,148.945
C06737=1214.926,-36.306,-40.382,-179.986,5.435,148.945
C06738=1214.930,-36.557,-40.369,-179.988,5.435,148.946
C06739=1214.935,-36.806,-40.357,-179.990,5.435,148.947
C06740=1214.941,-37.056,-40.345,-179.993,5.434,148.947
C06741=1214.945,-37.306,-40.332,-179.995,5.434,148.948
C06742=1214.951,-37.555,-40.319,-179.997,5.434,148.949
C06743=1214.956,-37.805,-40.306,-180.000,5.434,148.949
C06744=1214.961,-38.054,-40.293,179.997,5.433,148.950
C06745=1214.967,-38.303,-40.281,179.995,5.434,148.951
C06746=1214.971,-38.554,-40.269,179.993,5.433,148.952
C06747=1214.977,-38.803,-40.256,179.990,5.433,148.952
C06748=1214.982,-39.053,-40.243,179.988,5.433,148.953
C06749=1214.987,-39.302,-40.231,179.985,5.433,148.954
C06750=1214.992,-39.552,-40.217,179.983,5.432,148.954
C06751=1214.997,-39.802,-40.205,179.980,5.432,148.955
C06752=1215.003,-40.052,-40.193,179.978,5.432,148.956
C06753=1215.008,-40.301,-40.180,179.975,5.431,148.956
C06754=1215.013,-40.550,-40.167,179.974,5.431,148.957
C06755=1215.017,-40.800,-40.155,179.971,5.431,148.958
C06756=1215.023,-41.050,-40.143,179.969,5.431,148.958
C06757=1215.028,-41.299,-40.130,179.966,5.431,148.959
C06758=1215.033,-41.549,-40.117,179.963,5.430,148.960
C06759=1215.038,-41.798,-40.105,179.961,5.431,148.960
C06760=1215.043,-42.049,-40.093,179.959,5.430,148.961
C06761=1215.048,-42.298,-40.080,179.956,5.430,148.962
C06762=1215.053,-42.547,-40.067,179.954,5.430,148.963
C06763=1215.059,-42.797,-40.055,179.951,5.430,148.963
C06764=1215.064,-43.047,-40.043,179.949,5.429,148.964
C06765=1215.068,-43.297,-40.030,179.947,5.429,148.965
C06766=1215.073,-43.546,-40.017,179.944,5.429,148.965
C06767=1215.079,-43.796,-40.005,179.941,5.428,148.966
C06768=1215.084,-44.045,-39.993,179.939,5.429,148.967
C06769=1215.089,-44.295,-39.980,179.936,5.428,148.967
C06770=1215.095,-44.544,-39.968,179.934,5.427,148.968
C06771=1215.100,-44.794,-39.956,179.932,5.428,148.969
C06772=1215.104,-45.044,-39.943,179.930,5.427,148.969
C06773=1215.110,-45.294,-39.931,179.927,5.428,148.970
C06774=1215.115,-45.543,-39.918,179.925,5.427,148.971
C06775=1215.120,-45.793,-39.906,179.922,5.427,148.971
C06776=1215.125,-46.042,-39.894,179.920,5.427,148.972
C06777=1215.130,-46.292,-39.881,179.917,5.427,148.973
C06778=1215.136,-46.542,-39.869,179.915,5.426,148.974
C06779=1215.140,-46.792,-39.856,179.913,5.426,148.974
C06780=1215.146,-47.042,-39.844,179.910,5.426,148.975
C06781=1215.151,-47.291,-39.832,179.907,5.426,148.976
C06782=1215.156,-47.541,-39.820,179.905,5.426,148.976
C06783=1215.161,-47.790,-39.807,179.903,5.425,148.977
C06784=1215.167,-48.039,-39.795,179.901,5.426,148.978
C06785=1215.172,-48.289,-39.783,179.898,5.425,148.978
C06786=1215.177,-48.559,-39.769,179.895,5.425,148.979
C06787=1215.183,-48.829,-39.757,179.892,5.424,148.980
C06788=1215.189,-49.099,-39.743,179.890,5.425,148.981
C06789=1215.194,-49.369,-39.729,179.888,5.424,148.981
C06790=1215.199,-49.619,-39.717,179.885,5.424,148.982
C06791=1215.204,-49.868,-39.705,179.883,5.424,148.983
C06792=1215.209,-50.118,-39.694,179.880,5.424,148.983
C06793=1215.214,-50.367,-39.681,179.878,5.423,148.984
C06794=1215.220,-50.617,-39.669,179.876,5.423,148.985
C06795=1215.225,-50.867,-39.657,179.873,5.423,148.985
C06796=1215.230,-51.116,-39.645,179.871,5.423,148.986
C06797=1215.235,-51.366,-39.632,179.868,5.423,148.987
C06798=1215.241,-51.616,-39.620,179.865,5.422,148.988
C06799=1215.246,-51.865,-39.609,179.864,5.422,148.988
C06800=1215.250,-52.115,-39.596,179.861,5.422,148.989
C06801=1215.256,-52.365,-39.584,179.859,5.421,148.989
C06802=1215.261,-52.615,-39.571,179.856,5.422,148.990
C06803=1215.266,-52.865,-39.560,179.854,5.421,148.991
C06804=1215.271,-53.114,-39.547,179.852,5.422,148.992
C06805=1215.276,-53.364,-39.536,179.849,5.421,148.992
C06806=1215.281,-53.613,-39.524,179.846,5.421,148.993
C06807=1215.286,-53.863,-39.511,179.844,5.421,148.994
C06808=1215.292,-54.113,-39.499,179.842,5.421,148.994
C06809=1215.297,-54.362,-39.488,179.840,5.421,148.995
C06810=1215.302,-54.612,-39.475,179.837,5.421,148.996
C06811=1215.307,-54.862,-39.463,179.834,5.420,148.997
C06812=1215.313,-55.112,-39.452,179.832,5.420,148.997
C06813=1215.318,-55.361,-39.439,179.830,5.420,148.998
C06814=1215.322,-55.610,-39.428,179.828,5.420,148.998
C06815=1215.328,-55.860,-39.415,179.825,5.419,148.999
C06816=1215.333,-56.110,-39.403,179.823,5.419,149.000
C06817=1215.338,-56.360,-39.391,179.820,5.419,149.001
C06818=1215.343,-56.609,-39.380,179.818,5.419,149.001
C06819=1215.348,-56.859,-39.367,179.815,5.418,149.002
C06820=1215.354,-57.109,-39.356,179.813,5.419,149.003
C06821=1215.359,-57.358,-39.344,179.810,5.418,149.003
C06822=1215.363,-57.607,-39.332,179.808,5.419,149.004
C06823=1215.369,-57.857,-39.320,179.806,5.418,149.005
C06824=1215.374,-58.107,-39.308,179.803,5.418,149.005
C06825=1215.379,-58.357,-39.297,179.801,5.418,149.006
C06826=1215.384,-58.606,-39.284,179.798,5.418,149.007
C06827=1215.390,-58.856,-39.272,179.797,5.418,149.007
C06828=1215.394,-59.106,-39.261,179.794,5.417,149.008
C06829=1215.400,-59.356,-39.249,179.792,5.417,149.009
C06830=1215.405,-59.605,-39.236,179.789,5.417,149.009
C06831=1215.410,-59.854,-39.225,179.787,5.417,149.010
C06832=1215.416,-60.104,-39.214,179.784,5.417,149.011
C06833=1215.421,-60.354,-39.202,179.782,5.416,149.012
C06834=1215.426,-60.604,-39.190,179.780,5.417,149.012
C06835=1215.431,-60.853,-39.178,179.777,5.416,149.013
C06836=1215.436,-61.103,-39.166,179.774,5.416,149.014
C06837=1215.441,-61.352,-39.155,179.772,5.416,149.014
C06838=1215.446,-61.602,-39.143,179.770,5.416,149.015
C06839=1215.452,-61.852,-39.131,179.768,5.416,149.016
C06840=1215.456,-62.102,-39.120,179.765,5.415,149.016
C06841=1215.462,-62.352,-39.108,179.763,5.415,149.017
C06842=1215.467,-62.601,-39.095,179.761,5.415,149.018
C06843=1215.472,-62.851,-39.084,179.758,5.415,149.018
C06844=1215.478,-63.100,-39.072,179.756,5.415,149.019
C06845=1215.482,-63.350,-39.061,179.753,5.415,149.020
C06846=1215.488,-63.600,-39.049,179.750,5.414,149.020
C06847=1215.493,-63.850,-39.037,179.748,5.414,149.021
C06848=1215.498,-64.099,-39.026,179.746,5.414,149.022
C06849=1215.503,-64.349,-39.014,179.744,5.414,149.023
C06850=1215.508,-64.599,-39.003,179.741,5.414,149.023
C06851=1215.514,-64.849,-38.991,179.739,5.414,149.024
C06852=1215.519,-65.098,-38.978,179.737,5.413,149.024
C06853=1215.524,-65.347,-38.967,179.734,5.413,149.025
C06854=1215.529,-65.597,-38.955,179.732,5.413,149.026
C06855=1215.534,-65.846,-38.944,179.729,5.413,149.027
C06856=1215.539,-66.096,-38.932,179.727,5.413,149.027
C06857=1215.544,-66.346,-38.921,179.725,5.413,149.028
C06858=1215.550,-66.596,-38.909,179.722,5.413,149.029
C06859=1215.555,-66.845,-38.898,179.720,5.413,149.029
C06860=1215.560,-67.095,-38.886,179.717,5.412,149.030
C06861=1215.565,-67.344,-38.875,179.715,5.413,149.031
C06862=1215.570,-67.594,-38.863,179.712,5.412,149.032
C06863=1215.576,-67.844,-38.851,179.711,5.412,149.032
C06864=1215.581,-68.094,-38.840,179.708,5.412,149.033
C06865=1215.587,-68.343,-38.828,179.706,5.412,149.033
C06866=1215.591,-68.593,-38.817,179.703,5.412,149.034
C06867=1215.597,-68.843,-38.805,179.701,5.411,149.035
C06868=1215.602,-69.093,-38.795,179.699,5.411,149.036
C06869=1215.607,-69.343,-38.783,179.696,5.411,149.036
C06870=1215.612,-69.593,-38.771,179.694,5.411,149.037
C06871=1215.617,-69.841,-38.761,179.691,5.411,149.038
C06872=1215.623,-70.091,-38.749,179.689,5.411,149.038
C06873=1215.627,-70.341,-38.737,179.686,5.411,149.039
C06874=1215.633,-70.591,-38.725,179.684,5.410,149.040
C06875=1215.637,-70.841,-38.714,179.682,5.410,149.040
C06876=1215.643,-71.090,-38.703,179.679,5.410,149.041
C06877=1215.648,-71.339,-38.691,179.677,5.410,149.042
C06878=1215.654,-71.589,-38.679,179.675,5.410,149.042
C06879=1215.659,-71.840,-38.669,179.673,5.410,149.043
C06880=1215.665,-72.089,-38.657,179.670,5.410,149.044
C06881=1215.669,-72.339,-38.646,179.667,5.409,149.045
C06882=1215.674,-72.588,-38.635,179.665,5.410,149.045
C06883=1215.679,-72.838,-38.623,179.663,5.409,149.046
C06884=1215.685,-73.087,-38.612,179.660,5.409,149.047
C06885=1215.690,-73.338,-38.601,179.658,5.409,149.047
C06886=1215.695,-73.587,-38.590,179.656,5.409,149.048
C06887=1215.701,-73.837,-38.578,179.653,5.409,149.049
C06888=1215.706,-74.086,-38.567,179.651,5.409,149.049
C06889=1215.710,-74.336,-38.555,179.649,5.408,149.050
C06890=1215.716,-74.607,-38.543,179.646,5.408,149.051
C06891=1215.722,-74.877,-38.531,179.644,5.408,149.051
C06892=1215.728,-75.148,-38.519,179.641,5.408,149.052
C06893=1215.733,-75.418,-38.506,179.638,5.408,149.053
C06894=1215.739,-75.668,-38.496,179.637,5.408,149.054
C06895=1215.744,-75.917,-38.485,179.634,5.407,149.054
C06896=1215.749,-76.167,-38.473,179.632,5.408,149.055
C06897=1215.754,-76.417,-38.461,179.629,5.407,149.056
C06898=1215.759,-76.667,-38.451,179.627,5.408,149.056
C06899=1215.765,-76.916,-38.439,179.624,5.407,149.057
C06900=1215.769,-77.166,-38.428,179.622,5.407,149.058
C06901=1215.775,-77.415,-38.417,179.620,5.407,149.058
C06902=1215.780,-77.666,-38.406,179.617,5.407,149.059
C06903=1215.785,-77.915,-38.395,179.615,5.407,149.060
C06904=1215.790,-78.164,-38.384,179.613,5.406,149.060
C06905=1215.796,-78.415,-38.373,179.611,5.407,149.061
C06906=1215.801,-78.664,-38.361,179.608,5.406,149.062
C06907=1215.806,-78.914,-38.350,179.606,5.406,149.063
C06908=1215.812,-79.164,-38.339,179.603,5.406,149.063
C06909=1215.817,-79.413,-38.328,179.600,5.406,149.064
C06910=1215.821,-79.663,-38.317,179.598,5.406,149.065
C06911=1215.827,-79.913,-38.306,179.596,5.406,149.065
C06912=1215.832,-80.163,-38.294,179.594,5.406,149.066
C06913=1215.837,-80.412,-38.283,179.591,5.405,149.067
C06914=1215.843,-80.662,-38.273,179.589,5.405,149.067
C06915=1215.847,-80.911,-38.262,179.587,5.405,149.068
C06916=1215.853,-81.162,-38.251,179.585,5.405,149.069
C06917=1215.858,-81.411,-38.240,179.582,5.405,149.069
C06918=1215.863,-81.660,-38.228,179.580,5.405,149.070
C06919=1215.869,-81.910,-38.218,179.577,5.405,149.071
C06920=1215.874,-82.160,-38.206,179.575,5.405,149.072
C06921=1215.879,-82.410,-38.196,179.572,5.405,149.072
C06922=1215.884,-82.659,-38.185,179.570,5.404,149.073
C06923=1215.889,-82.909,-38.174,179.568,5.404,149.073
C06924=1215.894,-83.159,-38.163,179.565,5.404,149.074
C06925=1215.900,-83.408,-38.151,179.563,5.404,149.075
C06926=1215.905,-83.658,-38.141,179.561,5.404,149.076
C06927=1215.910,-83.908,-38.129,179.559,5.404,149.076
C06928=1215.915,-84.158,-38.119,179.556,5.404,149.077
C06929=1215.920,-84.407,-38.108,179.554,5.404,149.078
C06930=1215.926,-84.657,-38.097,179.552,5.403,149.078
C06931=1215.931,-84.907,-38.086,179.550,5.404,149.079
C06932=1215.936,-85.157,-38.075,179.547,5.403,149.080
C06933=1215.941,-85.406,-38.064,179.545,5.404,149.080
C06934=1215.946,-85.656,-38.054,179.542,5.403,149.081
C06935=1215.952,-85.905,-38.043,179.540,5.403,149.082
C06936=1215.957,-86.156,-38.032,179.537,5.403,149.082
C06937=1215.962,-86.405,-38.020,179.535,5.403,149.083
C06938=1215.968,-86.655,-38.010,179.533,5.403,149.084
C06939=1215.972,-86.904,-37.999,179.530,5.402,149.084
C06940=1215.978,-87.154,-37.989,179.528,5.402,149.085
C06941=1215.983,-87.404,-37.978,179.526,5.402,149.086
C06942=1215.988,-87.653,-37.967,179.524,5.402,149.086
C06943=1215.993,-87.903,-37.957,179.521,5.402,149.087
C06944=1215.998,-88.153,-37.945,179.519,5.402,149.088
C06945=1216.004,-88.403,-37.935,179.516,5.402,149.089
C06946=1216.009,-88.653,-37.924,179.515,5.402,149.089
C06947=1216.015,-88.902,-37.913,179.512,5.401,149.090
C06948=1216.020,-89.152,-37.902,179.510,5.402,149.090
C06949=1216.025,-89.401,-37.892,179.507,5.401,149.091
C06950=1216.030,-89.651,-37.881,179.505,5.402,149.092
C06951=1216.035,-89.901,-37.871,179.502,5.401,149.093
C06952=1216.040,-90.151,-37.859,179.500,5.402,149.093
C06953=1216.046,-90.400,-37.849,179.498,5.401,149.094
C06954=1216.051,-90.650,-37.839,179.496,5.401,149.095
C06955=1216.056,-90.899,-37.828,179.493,5.401,149.095
C06956=1216.061,-91.150,-37.817,179.491,5.401,149.096
C06957=1216.066,-91.400,-37.807,179.489,5.401,149.097
C06958=1216.071,-91.649,-37.796,179.486,5.401,149.097
C06959=1216.077,-91.899,-37.785,179.484,5.401,149.098
C06960=1216.083,-92.149,-37.774,179.482,5.401,149.099
C06961=1216.087,-92.398,-37.763,179.480,5.400,149.099
C06962=1216.093,-92.648,-37.753,179.477,5.401,149.100
C06963=1216.098,-92.898,-37.742,179.475,5.400,149.101
C06964=1216.103,-93.147,-37.731,179.473,5.401,149.101
C06965=1216.108,-93.397,-37.721,179.470,5.400,149.102
C06966=1216.114,-93.647,-37.711,179.468,5.400,149.103
C06967=1216.119,-93.896,-37.700,179.466,5.400,149.103
C06968=1216.124,-94.146,-37.689,179.463,5.399,149.104
C06969=1216.130,-94.396,-37.679,179.461,5.400,149.105
C06970=1216.135,-94.646,-37.668,179.458,5.399,149.105
C06971=1216.140,-94.895,-37.658,179.456,5.400,149.106
C06972=1216.145,-95.146,-37.647,179.454,5.399,149.107
C06973=1216.151,-95.395,-37.637,179.451,5.399,149.108
C06974=1216.155,-95.645,-37.627,179.449,5.399,149.108
C06975=1216.160,-95.894,-37.616,179.447,5.399,149.109
C06976=1216.165,-96.144,-37.606,179.444,5.399,149.109
C06977=1216.171,-96.394,-37.596,179.442,5.399,149.110
C06978=1216.176,-96.643,-37.584,179.440,5.399,149.111
C06979=1216.181,-96.893,-37.574,179.438,5.399,149.112
C06980=1216.187,-97.143,-37.564,179.435,5.398,149.112
C06981=1216.192,-97.393,-37.553,179.433,5.398,149.113
C06982=1216.197,-97.642,-37.543,179.431,5.398,149.114
C06983=1216.202,-97.893,-37.533,179.429,5.398,149.114
C06984=1216.208,-98.142,-37.522,179.426,5.398,149.115
C06985=1216.213,-98.392,-37.511,179.424,5.398,149.116
C06986=1216.218,-98.641,-37.501,179.421,5.398,149.116
C06987=1216.224,-98.891,-37.491,179.420,5.398,149.117
C06988=1216.228,-99.141,-37.481,179.417,5.397,149.118
C06989=1216.234,-99.390,-37.470,179.415,5.398,149.118
C06990=1216.239,-99.641,-37.460,179.412,5.397,149.119
C06991=1216.244,-99.890,-37.450,179.410,5.398,149.120
C06992=1216.250,-100.140,-37.439,179.407,5.397,149.120
C06993=1216.255,-100.389,-37.428,179.406,5.397,149.121
C06994=1216.260,-100.661,-37.417,179.403,5.397,149.122
C06995=1216.266,-100.931,-37.406,179.400,5.398,149.123
C06996=1216.272,-101.203,-37.395,179.398,5.397,149.123
C06997=1216.278,-101.474,-37.384,179.395,5.397,149.124
C06998=1216.283,-101.724,-37.373,179.393,5.397,149.125
C06999=1216.288,-101.973,-37.364,179.391,5.396,149.125
C07000=1216.293,-102.223,-37.353,179.389,5.397,149.126
C07001=1216.299,-102.473,-37.343,179.386,5.396,149.127
C07002=1216.304,-102.723,-37.332,179.384,5.397,149.127
C07003=1216.309,-102.973,-37.322,179.381,5.396,149.128
C07004=1216.314,-103.222,-37.313,179.379,5.397,149.129
C07005=1216.319,-103.472,-37.302,179.378,5.397,149.129
C07006=1216.325,-103.722,-37.292,179.375,5.396,149.130
C07007=1216.330,-103.971,-37.282,179.373,5.397,149.131
C07008=1216.335,-104.222,-37.271,179.370,5.396,149.131
C07009=1216.340,-104.471,-37.261,179.368,5.397,149.132
C07010=1216.346,-104.720,-37.251,179.366,5.396,149.133
C07011=1216.351,-104.971,-37.241,179.364,5.396,149.133
C07012=1216.356,-105.220,-37.230,179.361,5.396,149.134
C07013=1216.362,-105.470,-37.220,179.359,5.396,149.135
C07014=1216.366,-105.720,-37.210,179.356,5.396,149.135
C07015=1216.372,-105.969,-37.200,179.354,5.396,149.136
C07016=1216.377,-106.219,-37.190,179.352,5.395,149.137
C07017=1216.382,-106.469,-37.179,179.350,5.396,149.137
C07018=1216.387,-106.718,-37.170,179.347,5.395,149.138
C07019=1216.393,-106.968,-37.160,179.345,5.396,149.139
C07020=1216.398,-107.219,-37.149,179.343,5.395,149.139
C07021=1216.403,-107.468,-37.140,179.341,5.395,149.140
C07022=1216.409,-107.717,-37.130,179.338,5.395,149.141
C07023=1216.414,-107.968,-37.119,179.336,5.395,149.141
C07024=1216.419,-108.217,-37.109,179.333,5.395,149.142
C07025=1216.424,-108.466,-37.099,179.331,5.395,149.143
C07026=1216.430,-108.716,-37.089,179.329,5.394,149.143
C07027=1216.435,-108.967,-37.079,179.327,5.395,149.144
C07028=1216.440,-109.216,-37.070,179.324,5.394,149.145
C07029=1216.445,-109.466,-37.059,179.322,5.395,149.145
C07030=1216.450,-109.716,-37.049,179.320,5.394,149.146
C07031=1216.456,-109.965,-37.039,179.318,5.394,149.147
C07032=1216.461,-110.215,-37.029,179.315,5.394,149.147
C07033=1216.467,-110.465,-37.019,179.313,5.394,149.148
C07034=1216.472,-110.715,-37.009,179.311,5.394,149.149
C07035=1216.477,-110.964,-36.999,179.309,5.394,149.150
C07036=1216.482,-111.214,-36.989,179.307,5.394,149.150
C07037=1216.488,-111.463,-36.979,179.304,5.394,149.151
C07038=1216.492,-111.714,-36.970,179.302,5.394,149.151
C07039=1216.498,-111.963,-36.959,179.300,5.394,149.152
C07040=1216.503,-112.213,-36.950,179.297,5.394,149.153
C07041=1216.508,-112.462,-36.940,179.295,5.393,149.153
C07042=1216.514,-112.713,-36.930,179.293,5.394,149.154
C07043=1216.519,-112.962,-36.920,179.290,5.393,149.155
C07044=1216.524,-113.212,-36.910,179.288,5.394,149.155
C07045=1216.530,-113.461,-36.900,179.286,5.393,149.156
C07046=1216.534,-113.712,-36.890,179.284,5.393,149.157
C07047=1216.540,-113.961,-36.880,179.281,5.393,149.157
C07048=1216.545,-114.211,-36.871,179.279,5.393,149.158
C07049=1216.551,-114.461,-36.861,179.277,5.393,149.159
C07050=1216.556,-114.710,-36.851,179.275,5.393,149.160
C07051=1216.561,-114.960,-36.841,179.272,5.392,149.160
C07052=1216.566,-115.210,-36.831,179.270,5.393,149.161
C07053=1216.571,-115.460,-36.822,179.268,5.393,149.161
C07054=1216.577,-115.709,-36.812,179.265,5.393,149.162
C07055=1216.583,-115.959,-36.801,179.264,5.393,149.163
C07056=1216.587,-116.209,-36.792,179.261,5.392,149.163
C07057=1216.593,-116.459,-36.782,179.259,5.393,149.164
C07058=1216.598,-116.709,-36.773,179.256,5.392,149.165
C07059=1216.603,-116.958,-36.763,179.254,5.393,149.166
C07060=1216.608,-117.207,-36.753,179.252,5.392,149.166
C07061=1216.614,-117.458,-36.744,179.250,5.392,149.167
C07062=1216.618,-117.708,-36.734,179.247,5.392,149.167
C07063=1216.624,-117.957,-36.724,179.245,5.392,149.168
C07064=1216.629,-118.207,-36.715,179.243,5.391,149.169
C07065=1216.635,-118.457,-36.704,179.241,5.392,149.169
C07066=1216.640,-118.706,-36.696,179.238,5.391,149.170
C07067=1216.646,-118.956,-36.685,179.236,5.392,149.171
C07068=1216.650,-119.206,-36.675,179.234,5.392,149.172
C07069=1216.656,-119.456,-36.666,179.232,5.391,149.172
C07070=1216.661,-119.705,-36.656,179.230,5.392,149.173
C07071=1216.667,-119.955,-36.647,179.227,5.391,149.173
C07072=1216.671,-120.205,-36.637,179.225,5.392,149.174
C07073=1216.677,-120.455,-36.628,179.223,5.391,149.175
C07074=1216.682,-120.704,-36.618,179.221,5.391,149.175
C07075=1216.687,-120.955,-36.608,179.218,5.391,149.176
C07076=1216.692,-121.204,-36.599,179.216,5.391,149.177
C07077=1216.698,-121.454,-36.589,179.214,5.390,149.177
C07078=1216.703,-121.704,-36.579,179.212,5.391,149.178
C07079=1216.709,-121.953,-36.569,179.209,5.390,149.179
C07080=1216.714,-122.203,-36.560,179.207,5.391,149.179
C07081=1216.719,-122.452,-36.550,179.205,5.391,149.180
C07082=1216.725,-122.702,-36.541,179.203,5.390,149.181
C07083=1216.729,-122.953,-36.532,179.201,5.391,149.181
C07084=1216.735,-123.202,-36.522,179.198,5.390,149.182
C07085=1216.740,-123.452,-36.513,179.196,5.390,149.183
C07086=1216.746,-123.702,-36.503,179.194,5.390,149.183
C07087=1216.751,-123.952,-36.494,179.192,5.390,149.184
C07088=1216.756,-124.201,-36.484,179.189,5.390,149.185
C07089=1216.761,-124.451,-36.475,179.187,5.390,149.185
C07090=1216.766,-124.700,-36.465,179.185,5.389,149.186
C07091=1216.772,-124.950,-36.456,179.183,5.390,149.187
C07092=1216.777,-125.200,-36.446,179.180,5.390,149.187
C07093=1216.782,-125.450,-36.437,179.178,5.389,149.188
C07094=1216.788,-125.700,-36.428,179.176,5.390,149.189
C07095=1216.792,-125.950,-36.418,179.173,5.389,149.189
C07096=1216.798,-126.200,-36.408,179.171,5.390,149.190
C07097=1216.804,-126.450,-36.399,179.169,5.389,149.190
C07098=1216.382,-126.460,-36.436,179.165,5.393,149.193
C07099=1216.376,-126.210,-36.445,179.167,5.393,149.192
C07100=1216.372,-125.960,-36.455,179.170,5.393,149.191
C07101=1216.366,-125.710,-36.464,179.172,5.393,149.191
C07102=1216.361,-125.461,-36.474,179.174,5.393,149.190
C07103=1216.356,-125.211,-36.483,179.176,5.393,149.189
C07104=1216.350,-124.961,-36.492,179.179,5.393,149.188
C07105=1216.345,-124.712,-36.502,179.180,5.393,149.188
C07106=1216.340,-124.462,-36.511,179.183,5.393,149.187
C07107=1216.334,-124.212,-36.521,179.185,5.393,149.187
C07108=1216.329,-123.962,-36.530,179.188,5.393,149.186
C07109=1216.324,-123.713,-36.540,179.189,5.393,149.185
C07110=1216.319,-123.462,-36.550,179.192,5.394,149.185
C07111=1216.314,-123.212,-36.558,179.194,5.393,149.184
C07112=1216.308,-122.963,-36.569,179.197,5.394,149.183
C07113=1216.303,-122.713,-36.578,179.198,5.394,149.183
C07114=1216.297,-122.464,-36.588,179.201,5.394,149.182
C07115=1216.292,-122.214,-36.597,179.203,5.394,149.181
C07116=1216.287,-121.964,-36.606,179.205,5.394,149.181
C07117=1216.281,-121.714,-36.616,179.207,5.394,149.180
C07118=1216.276,-121.465,-36.625,179.209,5.394,149.179
C07119=1216.271,-121.214,-36.635,179.212,5.394,149.179
C07120=1216.266,-120.965,-36.645,179.214,5.394,149.178
C07121=1216.260,-120.715,-36.654,179.216,5.395,149.177
C07122=1216.256,-120.466,-36.664,179.218,5.394,149.177
C07123=1216.250,-120.216,-36.674,179.221,5.395,149.176
C07124=1216.245,-119.966,-36.683,179.223,5.394,149.175
C07125=1216.239,-119.717,-36.693,179.225,5.395,149.175
C07126=1216.234,-119.467,-36.702,179.228,5.395,149.174
C07127=1216.229,-119.217,-36.713,179.230,5.395,149.173
C07128=1216.224,-118.967,-36.722,179.232,5.395,149.173
C07129=1216.218,-118.717,-36.732,179.234,5.395,149.172
C07130=1216.213,-118.467,-36.741,179.237,5.395,149.171
C07131=1216.207,-118.218,-36.751,179.239,5.395,149.171
C07132=1216.203,-117.969,-36.761,179.241,5.395,149.170
C07133=1216.197,-117.718,-36.770,179.243,5.395,149.169
C07134=1216.192,-117.468,-36.780,179.246,5.396,149.169
C07135=1216.187,-117.218,-36.790,179.248,5.395,149.168
C07136=1216.182,-116.969,-36.799,179.250,5.396,149.167
C07137=1216.176,-116.719,-36.809,179.252,5.395,149.167
C07138=1216.171,-116.470,-36.818,179.255,5.396,149.166
C07139=1216.166,-116.219,-36.829,179.257,5.396,149.165
C07140=1216.161,-115.970,-36.838,179.259,5.396,149.165
C07141=1216.155,-115.720,-36.848,179.262,5.396,149.164
C07142=1216.150,-115.470,-36.858,179.264,5.397,149.164
C07143=1216.145,-115.221,-36.868,179.266,5.396,149.163
C07144=1216.139,-114.970,-36.878,179.268,5.396,149.162
C07145=1216.135,-114.721,-36.887,179.271,5.396,149.161
C07146=1216.129,-114.472,-36.897,179.273,5.396,149.161
C07147=1216.123,-114.221,-36.907,179.275,5.397,149.160
C07148=1216.118,-113.972,-36.917,179.277,5.396,149.160
C07149=1216.113,-113.722,-36.927,179.280,5.397,149.159
C07150=1216.108,-113.473,-36.937,179.282,5.396,149.158
C07151=1216.102,-113.223,-36.946,179.284,5.397,149.157
C07152=1216.097,-112.973,-36.956,179.286,5.397,149.157
C07153=1216.093,-112.723,-36.966,179.289,5.397,149.156
C07154=1216.087,-112.473,-36.976,179.291,5.397,149.155
C07155=1216.082,-112.224,-36.986,179.293,5.397,149.155
C07156=1216.076,-111.974,-36.996,179.295,5.397,149.154
C07157=1216.071,-111.725,-37.006,179.298,5.398,149.154
C07158=1216.066,-111.475,-37.016,179.300,5.397,149.153
C07159=1216.060,-111.224,-37.025,179.303,5.398,149.152
C07160=1216.055,-110.975,-37.036,179.305,5.397,149.151
C07161=1216.050,-110.726,-37.045,179.307,5.398,149.151
C07162=1216.045,-110.475,-37.056,179.309,5.398,149.150
C07163=1216.039,-110.225,-37.065,179.311,5.397,149.149
C07164=1216.034,-109.976,-37.075,179.314,5.398,149.149
C07165=1216.029,-109.726,-37.086,179.316,5.397,149.148
C07166=1216.024,-109.476,-37.096,179.318,5.398,149.148
C07167=1216.019,-109.227,-37.105,179.320,5.398,149.147
C07168=1216.013,-108.977,-37.116,179.323,5.398,149.146
C07169=1216.008,-108.727,-37.125,179.325,5.398,149.145
C07170=1216.002,-108.477,-37.136,179.327,5.398,149.145
C07171=1215.997,-108.228,-37.145,179.329,5.398,149.144
C07172=1215.992,-107.978,-37.155,179.332,5.399,149.144
C07173=1215.987,-107.728,-37.166,179.334,5.398,149.143
C07174=1215.982,-107.479,-37.176,179.337,5.399,149.142
C07175=1215.976,-107.229,-37.186,179.339,5.398,149.141
C07176=1215.971,-106.979,-37.196,179.341,5.399,149.141
C07177=1215.965,-106.729,-37.206,179.343,5.399,149.140
C07178=1215.961,-106.480,-37.216,179.346,5.399,149.139
C07179=1215.956,-106.229,-37.226,179.348,5.399,149.139
C07180=1215.950,-105.980,-37.236,179.350,5.399,149.138
C07181=1215.944,-105.730,-37.247,179.352,5.399,149.137
C07182=1215.940,-105.480,-37.257,179.355,5.400,149.137
C07183=1215.935,-105.231,-37.267,179.357,5.399,149.136
C07184=1215.929,-104.981,-37.277,179.359,5.400,149.135
C07185=1215.924,-104.731,-37.287,179.361,5.399,149.135
C07186=1215.919,-104.482,-37.297,179.364,5.400,149.134
C07187=1215.913,-104.232,-37.307,179.366,5.400,149.133
C07188=1215.908,-103.982,-37.318,179.368,5.400,149.133
C07189=1215.903,-103.732,-37.328,179.370,5.400,149.132
C07190=1215.897,-103.483,-37.338,179.373,5.400,149.131
C07191=1215.893,-103.233,-37.348,179.375,5.400,149.131
C07192=1215.887,-102.983,-37.359,179.378,5.400,149.130
C07193=1215.882,-102.734,-37.369,179.380,5.400,149.129
C07194=1215.877,-102.484,-37.379,179.382,5.401,149.129
C07195=1215.871,-102.234,-37.389,179.384,5.400,149.128
C07196=1215.867,-101.984,-37.399,179.386,5.400,149.127
C07197=1215.861,-101.735,-37.410,179.389,5.400,149.127
C07198=1215.856,-101.485,-37.420,179.391,5.400,149.126
C07199=1215.851,-101.214,-37.431,179.394,5.400,149.125
C07200=1215.845,-100.942,-37.442,179.397,5.401,149.124
C07201=1215.839,-100.672,-37.453,179.399,5.400,149.124
C07202=1215.833,-100.400,-37.464,179.401,5.401,149.123
C07203=1215.828,-100.150,-37.475,179.403,5.400,149.122
C07204=1215.822,-99.900,-37.485,179.406,5.401,149.122
C07205=1215.817,-99.651,-37.495,179.408,5.401,149.121
C07206=1215.813,-99.401,-37.506,179.410,5.401,149.120
C07207=1215.807,-99.152,-37.516,179.412,5.401,149.120
C07208=1215.802,-98.902,-37.527,179.415,5.401,149.119
C07209=1215.797,-98.652,-37.537,179.417,5.401,149.118
C07210=1215.791,-98.403,-37.547,179.419,5.402,149.118
C07211=1215.786,-98.152,-37.558,179.421,5.401,149.117
C07212=1215.780,-97.903,-37.568,179.424,5.402,149.116
C07213=1215.775,-97.652,-37.579,179.426,5.402,149.116
C07214=1215.770,-97.404,-37.590,179.429,5.402,149.115
C07215=1215.765,-97.153,-37.600,179.431,5.402,149.114
C07216=1215.760,-96.904,-37.610,179.433,5.402,149.114
C07217=1215.755,-96.655,-37.620,179.435,5.402,149.113
C07218=1215.750,-96.404,-37.631,179.438,5.402,149.112
C07219=1215.744,-96.155,-37.641,179.440,5.402,149.112
C07220=1215.739,-95.905,-37.652,179.443,5.403,149.111
C07221=1215.734,-95.656,-37.662,179.445,5.403,149.110
C07222=1215.729,-95.405,-37.673,179.447,5.403,149.109
C07223=1215.723,-95.156,-37.683,179.450,5.403,149.109
C07224=1215.718,-94.906,-37.694,179.452,5.403,149.108
C07225=1215.713,-94.657,-37.705,179.454,5.403,149.108
C07226=1215.707,-94.407,-37.715,179.457,5.403,149.107
C07227=1215.702,-94.157,-37.725,179.459,5.404,149.106
C07228=1215.697,-93.907,-37.736,179.461,5.403,149.105
C07229=1215.692,-93.658,-37.747,179.463,5.404,149.105
C07230=1215.686,-93.408,-37.757,179.466,5.404,149.104
C07231=1215.681,-93.158,-37.768,179.468,5.404,149.103
C07232=1215.676,-92.908,-37.778,179.470,5.404,149.103
C07233=1215.671,-92.659,-37.789,179.473,5.404,149.102
C07234=1215.666,-92.409,-37.799,179.475,5.404,149.101
C07235=1215.661,-92.159,-37.810,179.478,5.404,149.101
C07236=1215.655,-91.910,-37.821,179.479,5.404,149.100
C07237=1215.650,-91.660,-37.831,179.482,5.405,149.099
C07238=1215.645,-91.410,-37.842,179.484,5.404,149.099
C07239=1215.640,-91.160,-37.852,179.487,5.405,149.098
C07240=1215.634,-90.911,-37.863,179.489,5.404,149.097
C07241=1215.629,-90.661,-37.874,179.492,5.405,149.097
C07242=1215.624,-90.411,-37.884,179.494,5.404,149.096
C07243=1215.619,-90.162,-37.895,179.496,5.405,149.095
C07244=1215.613,-89.912,-37.905,179.498,5.405,149.095
C07245=1215.608,-89.662,-37.917,179.501,5.405,149.094
C07246=1215.603,-89.412,-37.928,179.503,5.405,149.093
C07247=1215.597,-89.162,-37.938,179.505,5.405,149.093
C07248=1215.593,-88.913,-37.949,179.507,5.405,149.092
C07249=1215.587,-88.663,-37.960,179.510,5.405,149.091
C07250=1215.582,-88.413,-37.970,179.512,5.405,149.091
C07251=1215.577,-88.164,-37.981,179.514,5.406,149.090
C07252=1215.572,-87.914,-37.992,179.516,5.405,149.089
C07253=1215.567,-87.665,-38.003,179.519,5.406,149.089
C07254=1215.562,-87.415,-38.013,179.522,5.406,149.088
C07255=1215.557,-87.164,-38.024,179.524,5.406,149.087
C07256=1215.551,-86.915,-38.035,179.527,5.406,149.086
C07257=1215.546,-86.665,-38.046,179.529,5.406,149.086
C07258=1215.540,-86.416,-38.057,179.531,5.407,149.085
C07259=1215.535,-86.166,-38.067,179.533,5.406,149.085
C07260=1215.530,-85.917,-38.078,179.536,5.407,149.084
C07261=1215.525,-85.667,-38.089,179.538,5.407,149.083
C07262=1215.520,-85.417,-38.100,179.540,5.407,149.082
C07263=1215.514,-85.167,-38.111,179.542,5.407,149.082
C07264=1215.509,-84.917,-38.122,179.545,5.407,149.081
C07265=1215.504,-84.668,-38.132,179.547,5.407,149.080
C07266=1215.499,-84.418,-38.144,179.549,5.408,149.080
C07267=1215.494,-84.168,-38.154,179.551,5.407,149.079
C07268=1215.489,-83.919,-38.165,179.554,5.408,149.078
C07269=1215.483,-83.669,-38.176,179.556,5.407,149.078
C07270=1215.478,-83.420,-38.187,179.559,5.408,149.077
C07271=1215.473,-83.169,-38.198,179.562,5.408,149.076
C07272=1215.468,-82.920,-38.209,179.564,5.408,149.076
C07273=1215.462,-82.670,-38.219,179.566,5.408,149.075
C07274=1215.457,-82.420,-38.231,179.568,5.408,149.074
C07275=1215.452,-82.171,-38.243,179.571,5.409,149.074
C07276=1215.447,-81.921,-38.253,179.573,5.408,149.073
C07277=1215.442,-81.671,-38.264,179.575,5.409,149.072
C07278=1215.437,-81.421,-38.275,179.577,5.408,149.071
C07279=1215.431,-81.172,-38.286,179.580,5.409,149.071
C07280=1215.426,-80.922,-38.297,179.582,5.408,149.070
C07281=1215.421,-80.673,-38.308,179.585,5.409,149.069
C07282=1215.416,-80.423,-38.319,179.586,5.409,149.069
C07283=1215.410,-80.173,-38.330,179.589,5.409,149.068
C07284=1215.405,-79.924,-38.341,179.592,5.410,149.067
C07285=1215.400,-79.674,-38.352,179.594,5.409,149.067
C07286=1215.395,-79.424,-38.363,179.597,5.410,149.066
C07287=1215.389,-79.175,-38.374,179.599,5.410,149.065
C07288=1215.384,-78.925,-38.386,179.601,5.410,149.065
C07289=1215.379,-78.675,-38.396,179.603,5.410,149.064
C07290=1215.374,-78.425,-38.408,179.606,5.410,149.063
C07291=1215.369,-78.176,-38.419,179.608,5.410,149.063
C07292=1215.364,-77.926,-38.430,179.610,5.411,149.062
C07293=1215.358,-77.676,-38.442,179.612,5.410,149.061
C07294=1215.353,-77.427,-38.452,179.615,5.411,149.061
C07295=1215.348,-77.177,-38.463,179.618,5.411,149.060
C07296=1215.343,-76.927,-38.474,179.620,5.411,149.059
C07297=1215.337,-76.678,-38.486,179.623,5.411,149.058
C07298=1215.332,-76.427,-38.496,179.625,5.411,149.058
C07299=1215.327,-76.177,-38.508,179.627,5.411,149.057
C07300=1215.322,-75.929,-38.519,179.629,5.411,149.057
C07301=1215.317,-75.679,-38.531,179.632,5.412,149.056
C07302=1215.311,-75.428,-38.542,179.634,5.411,149.055
C07303=1215.307,-75.158,-38.554,179.636,5.412,149.054
C07304=1215.300,-74.888,-38.566,179.640,5.412,149.053
